KUKA KRL program: MyProgram_343().src

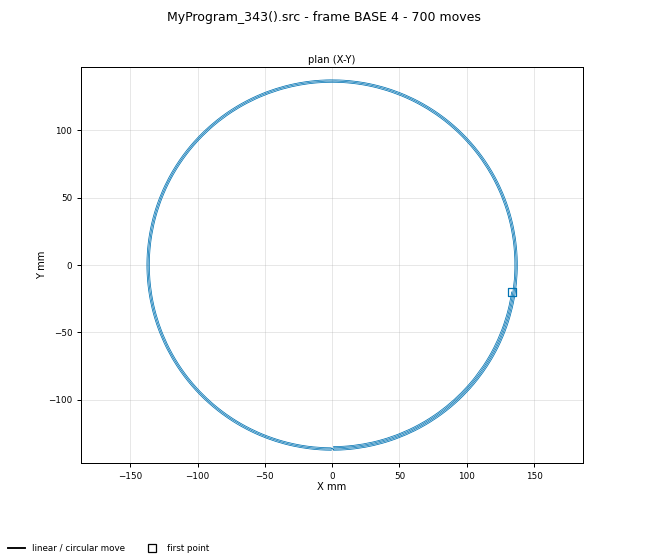
[picture p0: tool path of MyProgram_343().src in frame BASE 4, 700 of 700 moves have a stored position in this frame; points joined in program order, loops and branches not executed]
&ACCESS RVP
&REL 1
&PARAM TEMPLATE = C:\KRC\Roboter\Template\vorgabe
&PARAM EDITMASK = *
DEF MyProgram_343()
; ---- Setting reference (Base) ----
$BASE = BASE_DATA[4]

; --------------------------
; ---- Setting tool (TCP) ----
$TOOL = TOOL_DATA[3]
; --------------------------

$VEL.CP = VEL_APROX_PRINT
Startdeposition()
$VEL.CP = VEL_PRINT
LIN {X 133.4097,Y -19.9867,Z 192,A -2.4649,B 0.341,C 0.0391,E1 0.5017,E2 456.1576} C_DIS
LIN {X 132.7965,Y -23.712,Z 192,A -3.523,B 0.3407,C 0.0414,E1 0.5012,E2 457.1446} C_DIS
LIN {X 132.1464,Y -27.102,Z 192,A -4.5796,B 0.3404,C 0.0438,E1 0.5007,E2 458.1478} C_DIS
LIN {X 131.4928,Y -30.113,Z 192,A -5.5384,B 0.3401,C 0.0461,E1 0.5001,E2 459.0606} C_DIS
LIN {X 130.7303,Y -33.2675,Z 192,A -6.5628,B 0.3398,C 0.0485,E1 0.4994,E2 460.0383} C_DIS
LIN {X 129.6611,Y -37.224,Z 192,A -8.2205,B 0.3391,C 0.0529,E1 0.4982,E2 461.6861} C_DIS
LIN {X 128.1882,Y -42.0156,Z 192,A -9.2749,B 0.3388,C 0.0545,E1 0.4974,E2 462.5958} C_DIS
LIN {X 128.1882,Y -42.0156,Z 192,A -9.2759,B 0.3388,C 0.0545,E1 0.4974,E2 462.597} C_DIS
LIN {X 127.3782,Y -44.4067,Z 192,A -10.1216,B 0.3385,C 0.0565,E1 0.4967,E2 463.4123} C_DIS
LIN {X 126.1586,Y -47.7633,Z 192,A -11.2932,B 0.338,C 0.0593,E1 0.4956,E2 464.5374} C_DIS
LIN {X 124.0709,Y -52.952,Z 192,A -12.8743,B 0.3374,C 0.0626,E1 0.494,E2 466.01} C_DIS
LIN {X 123.0104,Y -55.3681,Z 192,A -13.7566,B 0.3371,C 0.0646,E1 0.493,E2 466.8596} C_DIS
LIN {X 121.4923,Y -58.6258,Z 192,A -14.8426,B 0.3366,C 0.067,E1 0.4918,E2 467.885} C_DIS
LIN {X 120.0893,Y -61.4469,Z 192,A -15.8424,B 0.3361,C 0.0692,E1 0.4906,E2 468.8379} C_DIS
LIN {X 118.1177,Y -65.1605,Z 192,A -17.0866,B 0.3356,C 0.0718,E1 0.489,E2 470.0066} C_DIS
LIN {X 116.3656,Y -68.2399,Z 192,A -18.2537,B 0.335,C 0.0745,E1 0.4874,E2 471.1268} C_DIS
LIN {X 114.2512,Y -71.7244,Z 192,A -19.5385,B 0.3344,C 0.0772,E1 0.4856,E2 472.3489} C_DIS
LIN {X 112.1427,Y -74.9777,Z 192,A -20.853,B 0.3337,C 0.0802,E1 0.4836,E2 473.6169} C_DIS
LIN {X 106.0971,Y -83.3128,Z 192,A -23.783,B 0.3323,C 0.0858,E1 0.479,E2 476.3404} C_DIS
LIN {X 106.0971,Y -83.3128,Z 192,A -23.7843,B 0.3323,C 0.0858,E1 0.479,E2 476.3418} C_DIS
LIN {X 104.2045,Y -85.6691,Z 192,A -25.3414,B 0.3312,C 0.09,E1 0.4761,E2 477.9401} C_DIS
LIN {X 100.7876,Y -89.6642,Z 192,A -26.4298,B 0.3308,C 0.0913,E1 0.4744,E2 478.862} C_DIS
LIN {X 95.9398,Y -94.8329,Z 192,A -28.8625,B 0.3294,C 0.0964,E1 0.4697,E2 481.2118} C_DIS
LIN {X 90.6247,Y -99.9239,Z 192,A -31.0205,B 0.3282,C 0.1003,E1 0.4655,E2 483.2275} C_DIS
LIN {X 90.6247,Y -99.9239,Z 192,A -31.0215,B 0.3282,C 0.1003,E1 0.4655,E2 483.2287} C_DIS
LIN {X 84.7075,Y -104.9869,Z 192,A -33.3755,B 0.3269,C 0.1046,E1 0.4607,E2 485.4418} C_DIS
LIN {X 81.036,Y -107.8465,Z 192,A -35.0547,B 0.3258,C 0.1079,E1 0.4569,E2 487.0775} C_DIS
LIN {X 78.9876,Y -109.3556,Z 192,A -35.9773,B 0.3252,C 0.1098,E1 0.4548,E2 487.9771} C_DIS
LIN {X 75.7275,Y -111.6377,Z 192,A -37.1784,B 0.3245,C 0.1118,E1 0.4521,E2 489.1052} C_DIS
LIN {X 72.4354,Y -113.8019,Z 192,A -38.5563,B 0.3236,C 0.1144,E1 0.4488,E2 490.4393} C_DIS
LIN {X 68.9662,Y -115.9366,Z 192,A -39.9703,B 0.3227,C 0.117,E1 0.4453,E2 491.8063} C_DIS
LIN {X 64.2775,Y -118.6008,Z 192,A -41.6506,B 0.3217,C 0.1197,E1 0.4413,E2 493.3947} C_DIS
LIN {X 60.7229,Y -120.4578,Z 192,A -42.8581,B 0.321,C 0.1215,E1 0.4383,E2 494.5271} C_DIS
LIN {X 57.4307,Y -122.0632,Z 192,A -44.0659,B 0.3202,C 0.1235,E1 0.4352,E2 495.6824} C_DIS
LIN {X 50.0734,Y -125.2593,Z 192,A -46.7069,B 0.3186,C 0.1276,E1 0.4283,E2 498.2071} C_DIS
LIN {X 50.0734,Y -125.2593,Z 192,A -46.7078,B 0.3186,C 0.1276,E1 0.4283,E2 498.2082} C_DIS
LIN {X 47.1757,Y -126.3787,Z 192,A -48.0353,B 0.3176,C 0.13,E1 0.4246,E2 499.5382} C_DIS
LIN {X 43.7279,Y -127.6136,Z 192,A -48.994,B 0.3172,C 0.131,E1 0.4222,E2 500.4049} C_DIS
LIN {X 40.7461,Y -128.5962,Z 192,A -50.0322,B 0.3166,C 0.1325,E1 0.4193,E2 501.398} C_DIS
LIN {X 37.4145,Y -129.6053,Z 192,A -51.21,B 0.3159,C 0.1342,E1 0.4161,E2 502.5299} C_DIS
LIN {X 34.0407,Y -130.5332,Z 192,A -52.5816,B 0.315,C 0.1363,E1 0.4121,E2 503.8847} C_DIS
LIN {X 29.855,Y -131.5518,Z 192,A -53.9027,B 0.3143,C 0.1379,E1 0.4085,E2 505.1273} C_DIS
LIN {X 26.0627,Y -132.3573,Z 192,A -55.1894,B 0.3136,C 0.1395,E1 0.4048,E2 506.3585} C_DIS
LIN {X 23.0754,Y -132.9104,Z 192,A -56.4574,B 0.3127,C 0.1414,E1 0.401,E2 507.6241} C_DIS
LIN {X 15.7245,Y -133.9776,Z 192,A -58.8527,B 0.3115,C 0.1441,E1 0.3942,E2 509.9018} C_DIS
LIN {X 11.9014,Y -134.3721,Z 192,A -60.2545,B 0.3107,C 0.1457,E1 0.39,E2 511.2683} C_DIS
LIN {X 8.165,Y -134.6498,Z 192,A -61.9084,B 0.3097,C 0.1479,E1 0.3849,E2 512.9333} C_DIS
LIN {X 3.8703,Y -134.8416,Z 192,A -63.1019,B 0.3093,C 0.1488,E1 0.3816,E2 514.0278} C_DIS
LIN {X 0.9691,Y -134.8866,Z 192,A -64.1734,B 0.3087,C 0.1499,E1 0.3784,E2 515.0745} C_DIS
Enddeposition()
LIN {X 0.9691,Y -134.8866,Z 192,A -64.1736,B 0.3087,C 0.1499,E1 0.3784,E2 515.0747} C_DIS
Startdeposition()
$VEL.CP = VEL_PRINT
LIN {X 1.4725,Y -135.79,Z 192,A -62.6899,B 0.3103,C 0.1468,E1 0.3836,E2 513.3947} C_DIS
LIN {X 7.8993,Y -135.5668,Z 192,A -61.1752,B 0.3106,C 0.1461,E1 0.3876,E2 512.0712} C_DIS
LIN {X 16.0493,Y -134.8442,Z 192,A -58.2123,B 0.3122,C 0.1426,E1 0.3964,E2 509.1841} C_DIS
LIN {X 22.9024,Y -133.8518,Z 192,A -55.8253,B 0.3135,C 0.1397,E1 0.4033,E2 506.8804} C_DIS
LIN {X 26.655,Y -133.1548,Z 192,A -54.5377,B 0.3143,C 0.1381,E1 0.407,E2 505.6431} C_DIS
LIN {X 31.7286,Y -132.037,Z 192,A -52.8298,B 0.3152,C 0.1359,E1 0.4118,E2 504.0106} C_DIS
LIN {X 34.8365,Y -131.2513,Z 192,A -51.7383,B 0.3159,C 0.1344,E1 0.4149,E2 502.9596} C_DIS
LIN {X 38.0279,Y -130.3624,Z 192,A -50.6047,B 0.3165,C 0.1328,E1 0.418,E2 501.8667} C_DIS
LIN {X 41.3599,Y -129.3438,Z 192,A -49.453,B 0.3172,C 0.1311,E1 0.4212,E2 500.7643} C_DIS
LIN {X 44.8211,Y -128.1859,Z 192,A -48.1394,B 0.3181,C 0.129,E1 0.4248,E2 499.4852} C_DIS
LIN {X 48.3933,Y -126.8826,Z 192,A -46.977,B 0.3187,C 0.1274,E1 0.4279,E2 498.3913} C_DIS
LIN {X 56.4469,Y -123.5092,Z 192,A -44.13,B 0.3204,C 0.123,E1 0.4353,E2 495.6732} C_DIS
LIN {X 56.4469,Y -123.5092,Z 192,A -44.131,B 0.3204,C 0.123,E1 0.4353,E2 495.6743} C_DIS
LIN {X 59.7456,Y -121.9467,Z 192,A -42.8805,B 0.3212,C 0.1209,E1 0.4385,E2 494.468} C_DIS
LIN {X 62.833,Y -120.3849,Z 192,A -41.7602,B 0.3219,C 0.1191,E1 0.4413,E2 493.3995} C_DIS
LIN {X 66.0403,Y -118.6581,Z 192,A -40.0165,B 0.3233,C 0.1153,E1 0.4459,E2 491.6221} C_DIS
LIN {X 71.1924,Y -115.6402,Z 192,A -38.6304,B 0.3239,C 0.1137,E1 0.4489,E2 490.4108} C_DIS
LIN {X 74.6132,Y -113.463,Z 192,A -37.2959,B 0.3247,C 0.1113,E1 0.452,E2 489.1331} C_DIS
LIN {X 77.4077,Y -111.5753,Z 192,A -36.1601,B 0.3254,C 0.1092,E1 0.4547,E2 488.0404} C_DIS
LIN {X 82.5823,Y -107.8014,Z 192,A -34.1686,B 0.3266,C 0.1057,E1 0.4591,E2 486.1562} C_DIS
LIN {X 85.9916,Y -105.1019,Z 192,A -32.4048,B 0.3278,C 0.1018,E1 0.463,E2 484.4018} C_DIS
LIN {X 89.8149,Y -101.8542,Z 192,A -31.1123,B 0.3284,C 0.0998,E1 0.4656,E2 483.2336} C_DIS
LIN {X 93.4233,Y -98.5553,Z 192,A -29.6342,B 0.3292,C 0.0971,E1 0.4685,E2 481.8427} C_DIS
LIN {X 96.6026,Y -95.4412,Z 192,A -28.4121,B 0.3299,C 0.095,E1 0.4708,E2 480.7182} C_DIS
LIN {X 100.2938,Y -91.5539,Z 192,A -26.5319,B 0.331,C 0.0909,E1 0.4744,E2 478.8935} C_DIS
LIN {X 104.4143,Y -86.8256,Z 192,A -24.5688,B 0.3321,C 0.087,E1 0.4779,E2 477.0305} C_DIS
LIN {X 106.2823,Y -84.5283,Z 192,A -23.3438,B 0.3328,C 0.084,E1 0.48,E2 475.8081} C_DIS
LIN {X 109.1526,Y -80.7877,Z 192,A -22.17,B 0.3333,C 0.082,E1 0.4818,E2 474.7539} C_DIS
LIN {X 113.2137,Y -74.9917,Z 192,A -19.9732,B 0.3344,C 0.0774,E1 0.4852,E2 472.6709} C_DIS
LIN {X 115.5535,Y -71.3337,Z 192,A -18.7754,B 0.3349,C 0.0751,E1 0.4868,E2 471.5643} C_DIS
LIN {X 117.7172,Y -67.7035,Z 192,A -17.3438,B 0.3357,C 0.0718,E1 0.4888,E2 470.1824} C_DIS
LIN {X 119.6857,Y -64.1585,Z 192,A -16.0569,B 0.3363,C 0.069,E1 0.4905,E2 468.9554} C_DIS
LIN {X 121.5238,Y -60.6031,Z 192,A -15.0058,B 0.3367,C 0.067,E1 0.4917,E2 467.9947} C_DIS
LIN {X 123.1566,Y -57.2094,Z 192,A -13.8117,B 0.3372,C 0.0643,E1 0.4931,E2 466.8557} C_DIS
LIN {X 124.7133,Y -53.7311,Z 192,A -12.1377,B 0.338,C 0.0597,E1 0.495,E2 465.1711} C_DIS
LIN {X 126.7888,Y -48.6353,Z 192,A -10.9268,B 0.3383,C 0.0578,E1 0.496,E2 464.1157} C_DIS
LIN {X 129.6598,Y -40.3634,Z 192,A -8.234,B 0.3393,C 0.0518,E1 0.4984,E2 461.5603} C_DIS
LIN {X 129.6598,Y -40.3634,Z 192,A -8.2351,B 0.3393,C 0.0518,E1 0.4984,E2 461.5615} C_DIS
LIN {X 130.6302,Y -37.1015,Z 192,A -7.1662,B 0.3397,C 0.0493,E1 0.4991,E2 460.5423} C_DIS
LIN {X 131.5427,Y -33.7207,Z 192,A -6.1536,B 0.34,C 0.047,E1 0.4998,E2 459.5926} C_DIS
LIN {X 132.3605,Y -30.351,Z 192,A -5.0792,B 0.3404,C 0.0445,E1 0.5005,E2 458.5702} C_DIS
LIN {X 133.111,Y -26.8701,Z 192,A -3.9875,B 0.3407,C 0.042,E1 0.5011,E2 457.5333} C_DIS
LIN {X 133.867,Y -22.8113,Z 192,A -2.6959,B 0.341,C 0.039,E1 0.5017,E2 456.3014} C_DIS
LIN {X 134.4202,Y -19.2804,Z 192,A -1.692,B 0.3413,C 0.0368,E1 0.5021,E2 455.3639} C_DIS
LIN {X 135.3511,Y -10.9921,Z 192,A 0.9276,B 0.3419,C 0.0306,E1 0.5028,E2 452.8614} C_DIS
LIN {X 135.5771,Y -7.7314,Z 192,A 2.3132,B 0.3422,C 0.0267,E1 0.503,E2 451.4743} C_DIS
LIN {X 135.7734,Y -2.4939,Z 192,A 3.3682,B 0.3423,C 0.0251,E1 0.503,E2 450.5685} C_DIS
LIN {X 135.7363,Y 4.038,Z 192,A 5.4733,B 0.3427,C 0.0199,E1 0.503,E2 448.5455} C_DIS
LIN {X 135.5506,Y 8.1615,Z 192,A 6.7874,B 0.3428,C 0.0167,E1 0.5028,E2 447.2848} C_DIS
LIN {X 135.0975,Y 13.7679,Z 192,A 8.6876,B 0.343,C 0.0119,E1 0.5023,E2 445.443} C_DIS
LIN {X 134.622,Y 17.8179,Z 192,A 9.6568,B 0.3431,C 0.0101,E1 0.502,E2 444.5665} C_DIS
LIN {X 133.9777,Y 22.1475,Z 192,A 10.9665,B 0.3431,C 0.007,E1 0.5015,E2 443.322} C_DIS
LIN {X 133.1461,Y 26.6974,Z 192,A 12.3466,B 0.3432,C 0.0037,E1 0.5008,E2 442.0106} C_DIS
LIN {X 132.4245,Y 30.0708,Z 192,A 13.3988,B 0.3432,C 0.0013,E1 0.5002,E2 441.0063} C_DIS
LIN {X 131.5924,Y 33.5252,Z 192,A 14.4549,B 0.3432,C -0.0012,E1 0.4995,E2 440.0026} C_DIS
LIN {X 130.641,Y 37.0629,Z 192,A 15.6611,B 0.3432,C -0.0042,E1 0.4986,E2 438.8361} C_DIS
LIN {X 129.434,Y 41.0773,Z 192,A 16.8602,B 0.3432,C -0.0069,E1 0.4977,E2 437.7032} C_DIS
LIN {X 128.3363,Y 44.3873,Z 192,A 17.8557,B 0.3432,C -0.0091,E1 0.4968,E2 436.7624} C_DIS
LIN {X 125.7972,Y 51.1436,Z 192,A 20.1438,B 0.3429,C -0.0146,E1 0.4946,E2 434.5603} C_DIS
LIN {X 124.4817,Y 54.2669,Z 192,A 21.546,B 0.3428,C -0.0184,E1 0.493,E2 433.1609} C_DIS
LIN {X 122.3912,Y 58.8295,Z 192,A 22.6661,B 0.3426,C -0.0204,E1 0.4918,E2 432.1522} C_DIS
LIN {X 120.4119,Y 62.7817,Z 192,A 23.9979,B 0.3425,C -0.0235,E1 0.4902,E2 430.8788} C_DIS
LIN {X 118.3975,Y 66.5056,Z 192,A 25.2069,B 0.3423,C -0.0262,E1 0.4886,E2 429.7323} C_DIS
LIN {X 115.3361,Y 71.6837,Z 192,A 27.0194,B 0.3419,C -0.0302,E1 0.4861,E2 427.9972} C_DIS
LIN {X 115.3361,Y 71.6837,Z 192,A 27.0182,B 0.3419,C -0.0302,E1 0.4861,E2 427.9986} C_DIS
LIN {X 111.0879,Y 78.1055,Z 192,A 29.5384,B 0.3413,C -0.0361,E1 0.4823,E2 425.5547} C_DIS
LIN {X 111.0879,Y 78.1055,Z 192,A 29.5372,B 0.3413,C -0.0361,E1 0.4823,E2 425.556} C_DIS
LIN {X 108.4803,Y 81.6884,Z 192,A 30.8927,B 0.341,C -0.0392,E1 0.48,E2 424.2536} C_DIS
LIN {X 105.7497,Y 85.1937,Z 192,A 32.2508,B 0.3407,C -0.0422,E1 0.4777,E2 422.948} C_DIS
LIN {X 102.9151,Y 88.5971,Z 192,A 33.6229,B 0.3403,C -0.0452,E1 0.4753,E2 421.6259} C_DIS
LIN {X 99.8987,Y 91.9849,Z 192,A 35.0225,B 0.3398,C -0.0483,E1 0.4727,E2 420.2773} C_DIS
LIN {X 96.841,Y 95.1987,Z 192,A 36.3962,B 0.3394,C -0.0512,E1 0.47,E2 418.9523} C_DIS
LIN {X 93.6737,Y 98.317,Z 192,A 37.7131,B 0.339,C -0.054,E1 0.4674,E2 417.6895} C_DIS
LIN {X 90.8265,Y 100.9534,Z 192,A 39.0052,B 0.3385,C -0.0568,E1 0.4647,E2 416.4302} C_DIS
LIN {X 87.3782,Y 103.952,Z 192,A 40.4055,B 0.338,C -0.0597,E1 0.4618,E2 415.0798} C_DIS
LIN {X 83.9483,Y 106.741,Z 192,A 41.7906,B 0.3375,C -0.0625,E1 0.4587,E2 413.7393} C_DIS
LIN {X 80.4014,Y 109.4375,Z 192,A 43.1692,B 0.337,C -0.0653,E1 0.4556,E2 412.4066} C_DIS
LIN {X 76.908,Y 111.9202,Z 192,A 44.5345,B 0.3364,C -0.068,E1 0.4524,E2 411.0814} C_DIS
LIN {X 70.7158,Y 115.9326,Z 192,A 47.4997,B 0.3351,C -0.0744,E1 0.4451,E2 408.1298} C_DIS
LIN {X 64.99,Y 119.2362,Z 192,A 48.9607,B 0.3346,C -0.0765,E1 0.4417,E2 406.7851} C_DIS
LIN {X 64.99,Y 119.2362,Z 192,A 48.9597,B 0.3346,C -0.0765,E1 0.4417,E2 406.7862} C_DIS
LIN {X 61.8234,Y 120.9063,Z 192,A 50.0685,B 0.3341,C -0.0786,E1 0.4388,E2 405.7115} C_DIS
LIN {X 58.7094,Y 122.4486,Z 192,A 51.1303,B 0.3337,C -0.0805,E1 0.4361,E2 404.6839} C_DIS
LIN {X 55.145,Y 124.0949,Z 192,A 52.7437,B 0.3329,C -0.0837,E1 0.4318,E2 403.0743} C_DIS
LIN {X 51.4888,Y 125.658,Z 192,A 53.7858,B 0.3325,C -0.0853,E1 0.429,E2 402.0849} C_DIS
LIN {X 44.4612,Y 128.3107,Z 192,A 56.2033,B 0.3314,C -0.0894,E1 0.4225,E2 399.7283} C_DIS
LIN {X 40.3327,Y 129.6692,Z 192,A 57.6658,B 0.3307,C -0.0918,E1 0.4183,E2 398.2954} C_DIS
LIN {X 36.6706,Y 130.7507,Z 192,A 58.8285,B 0.3302,C -0.0936,E1 0.4151,E2 397.1677} C_DIS
LIN {X 33.7939,Y 131.5242,Z 192,A 59.8669,B 0.3298,C -0.0953,E1 0.4121,E2 396.1463} C_DIS
LIN {X 30.415,Y 132.3459,Z 192,A 61.0053,B 0.3293,C -0.097,E1 0.4088,E2 395.0332} C_DIS
LIN {X 27.1208,Y 133.06,Z 192,A 62.1582,B 0.3287,C -0.0988,E1 0.4055,E2 393.9007} C_DIS
LIN {X 23.1296,Y 133.8139,Z 192,A 63.4762,B 0.3282,C -0.1006,E1 0.4016,E2 392.6126} C_DIS
LIN {X 18.7384,Y 134.4976,Z 192,A 65.0518,B 0.3275,C -0.1029,E1 0.397,E2 391.0593} C_DIS
LIN {X 14.8354,Y 134.9835,Z 192,A 66.3029,B 0.327,C -0.1045,E1 0.3933,E2 389.838} C_DIS
LIN {X 11.464,Y 135.3112,Z 192,A 67.7711,B 0.3263,C -0.1066,E1 0.3888,E2 388.3675} C_DIS
LIN {X 8.0751,Y 135.556,Z 192,A 69.1287,B 0.3257,C -0.1084,E1 0.3847,E2 387.0158} C_DIS
LIN {X 3.576,Y 135.7491,Z 192,A 70.2654,B 0.3253,C -0.1095,E1 0.3813,E2 385.9331} C_DIS
LIN {X 0.1229,Y 135.7975,Z 192,A 71.9806,B 0.3246,C -0.1118,E1 0.376,E2 384.2007} C_DIS
LIN {X -4.7497,Y 135.714,Z 192,A 73.1804,B 0.3242,C -0.1128,E1 0.3725,E2 383.0603} C_DIS
LIN {X -11.1773,Y 135.3354,Z 192,A 75.4863,B 0.3234,C -0.1151,E1 0.3655,E2 380.7826} C_DIS
LIN {X -11.1773,Y 135.3354,Z 192,A 75.4853,B 0.3234,C -0.1151,E1 0.3655,E2 380.7837} C_DIS
LIN {X -14.4957,Y 135.02,Z 192,A 76.7242,B 0.323,C -0.1163,E1 0.3616,E2 379.5564} C_DIS
LIN {X -18.0871,Y 134.5867,Z 192,A 78.2157,B 0.3225,C -0.1176,E1 0.357,E2 378.0679} C_DIS
LIN {X -23.7428,Y 133.7042,Z 192,A 80.1421,B 0.3219,C -0.1191,E1 0.3512,E2 376.1739} C_DIS
LIN {X -26.8096,Y 133.1233,Z 192,A 81.2932,B 0.3216,C -0.1199,E1 0.3477,E2 375.034} C_DIS
LIN {X -30.1125,Y 132.415,Z 192,A 82.5489,B 0.3213,C -0.1208,E1 0.3439,E2 373.7895} C_DIS
LIN {X -33.0981,Y 131.7008,Z 192,A 83.7349,B 0.321,C -0.1215,E1 0.3403,E2 372.611} C_DIS
LIN {X -36.3353,Y 130.8445,Z 192,A 85.0496,B 0.3207,C -0.1223,E1 0.3364,E2 371.303} C_DIS
LIN {X -39.8506,Y 129.8168,Z 192,A 86.3814,B 0.3205,C -0.1229,E1 0.3324,E2 369.985} C_DIS
LIN {X -47.1065,Y 127.3645,Z 192,A 89.4772,B 0.32,C -0.1242,E1 0.3232,E2 366.8992} C_DIS
LIN {X -50.5062,Y 126.0541,Z 192,A 90.8198,B 0.3199,C -0.1245,E1 0.3193,E2 365.5691} C_DIS
LIN {X -53.4792,Y 124.8223,Z 192,A 92.1446,B 0.3197,C -0.1249,E1 0.3155,E2 364.2468} C_DIS
LIN {X -56.5005,Y 123.4844,Z 192,A 93.6692,B 0.3197,C -0.1252,E1 0.3111,E2 362.715} C_DIS
LIN {X -60.1379,Y 121.7532,Z 192,A 95.1103,B 0.3196,C -0.1252,E1 0.307,E2 361.2902} C_DIS
LIN {X -62.8614,Y 120.37,Z 192,A 96.4981,B 0.3196,C -0.1253,E1 0.3031,E2 359.897} C_DIS
LIN {X -65.1407,Y 119.154,Z 192,A 98.2018,B 0.3196,C -0.1254,E1 0.2983,E2 358.1562} C_DIS
LIN {X -69.1565,Y 116.8697,Z 192,A 100.5286,B 0.3196,C -0.1252,E1 0.2919,E2 355.8066} C_DIS
LIN {X -74.392,Y 113.6086,Z 192,A 102.4653,B 0.3199,C -0.1244,E1 0.2869,E2 353.9127} C_DIS
LIN {X -78.1055,Y 111.0879,Z 192,A 104.3444,B 0.3202,C -0.1238,E1 0.282,E2 352.0353} C_DIS
LIN {X -84.2675,Y 106.4898,Z 192,A 108.0185,B 0.3208,C -0.1221,E1 0.2728,E2 348.3361} C_DIS
LIN {X -87.7024,Y 103.6791,Z 192,A 110.1144,B 0.3213,C -0.1208,E1 0.2677,E2 346.227} C_DIS
LIN {X -90.5619,Y 101.1904,Z 192,A 112.1309,B 0.3218,C -0.1194,E1 0.2629,E2 344.1846} C_DIS
LIN {X -96.1175,Y 95.9295,Z 192,A 115.7507,B 0.323,C -0.1163,E1 0.2547,E2 340.5407} C_DIS
LIN {X -99.6018,Y 92.3068,Z 192,A 118.9115,B 0.324,C -0.1133,E1 0.2479,E2 337.3112} C_DIS
LIN {X -102.7604,Y 88.7767,Z 192,A 121.1506,B 0.3249,C -0.1107,E1 0.2433,E2 335.0564} C_DIS
LIN {X -105.1673,Y 85.9115,Z 192,A 122.7645,B 0.3256,C -0.1087,E1 0.2402,E2 333.4407} C_DIS
LIN {X -107.9808,Y 82.3477,Z 192,A 125.1208,B 0.3266,C -0.1056,E1 0.2357,E2 331.0545} C_DIS
LIN {X -110.4857,Y 78.9549,Z 192,A 127.5551,B 0.3277,C -0.1022,E1 0.2312,E2 328.5741} C_DIS
LIN {X -112.8828,Y 75.4881,Z 192,A 130.0053,B 0.3288,C -0.0986,E1 0.227,E2 326.0753} C_DIS
LIN {X -115.39,Y 71.5971,Z 192,A 132.5678,B 0.33,C -0.0945,E1 0.2228,E2 323.4679} C_DIS
LIN {X -117.9533,Y 67.2903,Z 192,A 135.6435,B 0.3314,C -0.0893,E1 0.218,E2 320.3187} C_DIS
LIN {X -117.9533,Y 67.2903,Z 192,A 135.6426,B 0.3314,C -0.0893,E1 0.218,E2 320.3197} C_DIS
LIN {X -119.8647,Y 63.8237,Z 192,A 138.2995,B 0.3327,C -0.0846,E1 0.2141,E2 317.5845} C_DIS
LIN {X -119.8647,Y 63.8237,Z 192,A 138.2983,B 0.3327,C -0.0846,E1 0.2141,E2 317.5858} C_DIS
LIN {X -121.8013,Y 60.0404,Z 192,A 140.6505,B 0.3338,C -0.0801,E1 0.2109,E2 315.1883} C_DIS
LIN {X -123.2085,Y 57.0972,Z 192,A 142.6988,B 0.3347,C -0.0761,E1 0.2083,E2 313.0841} C_DIS
LIN {X -124.9738,Y 53.1288,Z 192,A 145.7,B 0.336,C -0.07,E1 0.2047,E2 309.9827} C_DIS
LIN {X -124.9738,Y 53.1288,Z 192,A 145.6985,B 0.336,C -0.07,E1 0.2047,E2 309.9843} C_DIS
LIN {X -126.4123,Y 49.6038,Z 192,A 148.0693,B 0.3371,C -0.0649,E1 0.202,E2 307.546} C_DIS
LIN {X -127.7059,Y 46.1697,Z 192,A 150.5189,B 0.338,C -0.0596,E1 0.1995,E2 305.0146} C_DIS
LIN {X -127.7059,Y 46.1697,Z 192,A 150.5179,B 0.338,C -0.0596,E1 0.1995,E2 305.0157} C_DIS
LIN {X -128.8341,Y 42.9211,Z 192,A 152.7094,B 0.3389,C -0.0547,E1 0.1974,E2 302.7555} C_DIS
LIN {X -129.8022,Y 39.8984,Z 192,A 154.9878,B 0.3397,C -0.0494,E1 0.1953,E2 300.3876} C_DIS
LIN {X -129.8022,Y 39.8984,Z 192,A 154.9867,B 0.3397,C -0.0494,E1 0.1953,E2 300.3888} C_DIS
LIN {X -130.7106,Y 36.8139,Z 192,A 157.2197,B 0.3404,C -0.0442,E1 0.1935,E2 298.0703} C_DIS
LIN {X -130.7106,Y 36.8139,Z 192,A 157.2187,B 0.3404,C -0.0442,E1 0.1935,E2 298.0714} C_DIS
LIN {X -131.6889,Y 33.1448,Z 192,A 160.4515,B 0.3413,C -0.0365,E1 0.1911,E2 294.6736} C_DIS
LIN {X -132.445,Y 29.9813,Z 192,A 162.4614,B 0.3418,C -0.0316,E1 0.1898,E2 292.5976} C_DIS
LIN {X -132.445,Y 29.9813,Z 192,A 162.4597,B 0.3418,C -0.0316,E1 0.1898,E2 292.5995} C_DIS
LIN {X -133.33,Y 25.7622,Z 192,A 165.3538,B 0.3424,C -0.0243,E1 0.1881,E2 289.5915} C_DIS
LIN {X -133.33,Y 25.7622,Z 192,A 165.3524,B 0.3424,C -0.0243,E1 0.1881,E2 289.5931} C_DIS
LIN {X -133.8722,Y 22.7799,Z 192,A 167.7024,B 0.3428,C -0.0184,E1 0.1869,E2 287.1263} C_DIS
LIN {X -133.8722,Y 22.7799,Z 192,A 167.7005,B 0.3428,C -0.0184,E1 0.1869,E2 287.1284} C_DIS
LIN {X -134.4634,Y 18.9781,Z 192,A 170.4332,B 0.3431,C -0.0114,E1 0.1857,E2 284.2721} C_DIS
LIN {X -134.4634,Y 18.9781,Z 192,A 170.4315,B 0.3431,C -0.0114,E1 0.1857,E2 284.2739} C_DIS
LIN {X -134.9487,Y 15.1585,Z 192,A 173.4823,B 0.3432,C -0.0036,E1 0.1847,E2 281.0595} C_DIS
LIN {X -134.9487,Y 15.1585,Z 192,A 173.4795,B 0.3432,C -0.0036,E1 0.1847,E2 281.0626} C_DIS
LIN {X -135.3338,Y 11.1966,Z 192,A 176.3421,B 0.3432,C 0.0038,E1 0.1839,E2 278.0606} C_DIS
LIN {X -135.3338,Y 11.1966,Z 192,A 176.34,B 0.3432,C 0.0038,E1 0.1839,E2 278.063} C_DIS
LIN {X -135.6201,Y 6.9103,Z 192,A 179.4355,B 0.343,C 0.0119,E1 0.1834,E2 274.8127} C_DIS
LIN {X -135.6201,Y 6.9103,Z 192,A 179.4334,B 0.343,C 0.0119,E1 0.1834,E2 274.815} C_DIS
LIN {X -135.7595,Y 3.2026,Z 192,A -177.5746,B 0.3427,C 0.0197,E1 0.1831,E2 271.6464} C_DIS
LIN {X -135.7595,Y 3.2026,Z 192,A -177.5775,B 0.3427,C 0.0197,E1 0.1831,E2 271.6497} C_DIS
LIN {X -135.7975,Y -0.3872,Z 192,A -174.886,B 0.3422,C 0.0267,E1 0.1831,E2 268.8092} C_DIS
LIN {X -135.7975,Y -0.3872,Z 192,A -174.8886,B 0.3422,C 0.0267,E1 0.1831,E2 268.8122} C_DIS
LIN {X -135.7197,Y -4.6055,Z 192,A -171.8245,B 0.3415,C 0.0347,E1 0.1834,E2 265.5821} C_DIS
LIN {X -135.7197,Y -4.6055,Z 192,A -171.8269,B 0.3415,C 0.0347,E1 0.1834,E2 265.5847} C_DIS
LIN {X -135.5466,Y -8.2274,Z 192,A -169.3151,B 0.3408,C 0.0412,E1 0.1837,E2 262.9438} C_DIS
LIN {X -135.5466,Y -8.2274,Z 192,A -169.3164,B 0.3408,C 0.0412,E1 0.1837,E2 262.9452} C_DIS
LIN {X -135.3293,Y -11.2493,Z 192,A -166.9224,B 0.34,C 0.0473,E1 0.1843,E2 260.4019} C_DIS
LIN {X -135.3293,Y -11.2493,Z 192,A -166.9241,B 0.34,C 0.0473,E1 0.1843,E2 260.4038} C_DIS
LIN {X -134.9468,Y -15.1761,Z 192,A -163.8815,B 0.3388,C 0.055,E1 0.1853,E2 257.1734} C_DIS
LIN {X -134.9468,Y -15.1761,Z 192,A -163.884,B 0.3388,C 0.055,E1 0.1853,E2 257.1763} C_DIS
LIN {X -134.4347,Y -19.1791,Z 192,A -161.193,B 0.3377,C 0.0618,E1 0.1863,E2 254.3486} C_DIS
LIN {X -134.4347,Y -19.1791,Z 192,A -161.1942,B 0.3377,C 0.0618,E1 0.1863,E2 254.35} C_DIS
LIN {X -133.9536,Y -22.2921,Z 192,A -158.8015,B 0.3365,C 0.0676,E1 0.1875,E2 251.8079} C_DIS
LIN {X -133.9536,Y -22.2921,Z 192,A -158.8029,B 0.3365,C 0.0676,E1 0.1875,E2 251.8095} C_DIS
LIN {X -133.2691,Y -26.0805,Z 192,A -155.9622,B 0.3351,C 0.0744,E1 0.189,E2 248.7957} C_DIS
LIN {X -133.2691,Y -26.0805,Z 192,A -155.964,B 0.3351,C 0.0744,E1 0.189,E2 248.7978} C_DIS
LIN {X -132.4319,Y -30.0387,Z 192,A -153.3172,B 0.3336,C 0.0807,E1 0.1907,E2 246.0156} C_DIS
LIN {X -132.4319,Y -30.0387,Z 192,A -153.3182,B 0.3336,C 0.0807,E1 0.1907,E2 246.0168} C_DIS
LIN {X -131.6604,Y -33.2572,Z 192,A -150.9302,B 0.3322,C 0.0862,E1 0.1924,E2 243.4842} C_DIS
LIN {X -131.6604,Y -33.2572,Z 192,A -150.9312,B 0.3322,C 0.0862,E1 0.1924,E2 243.4854} C_DIS
LIN {X -130.6807,Y -36.9208,Z 192,A -148.264,B 0.3306,C 0.0922,E1 0.1946,E2 240.6609} C_DIS
LIN {X -130.6807,Y -36.9208,Z 192,A -148.2651,B 0.3306,C 0.0922,E1 0.1946,E2 240.6623} C_DIS
LIN {X -129.4697,Y -40.9657,Z 192,A -145.6057,B 0.3289,C 0.0981,E1 0.1969,E2 237.8724} C_DIS
LIN {X -128.5394,Y -43.8017,Z 192,A -143.0028,B 0.3273,C 0.1034,E1 0.1995,E2 235.0672} C_DIS
LIN {X -128.5394,Y -43.8017,Z 192,A -143.005,B 0.3273,C 0.1034,E1 0.1995,E2 235.0697} C_DIS
LIN {X -126.5814,Y -49.1688,Z 192,A -139.6955,B 0.3251,C 0.1102,E1 0.203,E2 231.6239} C_DIS
LIN {X -125.379,Y -52.1589,Z 192,A -137.6043,B 0.3237,C 0.1143,E1 0.2055,E2 229.4209} C_DIS
LIN {X -124.0007,Y -55.3557,Z 192,A -135.3447,B 0.3221,C 0.1185,E1 0.2083,E2 227.0397} C_DIS
LIN {X -122.6394,Y -58.3099,Z 192,A -133.3866,B 0.3208,C 0.1221,E1 0.2108,E2 224.9911} C_DIS
LIN {X -121.1396,Y -61.365,Z 192,A -131.3757,B 0.3194,C 0.1256,E1 0.2136,E2 222.8909} C_DIS
LIN {X -118.5397,Y -66.2526,Z 192,A -127.8127,B 0.3171,C 0.1314,E1 0.2189,E2 219.136} C_DIS
LIN {X -118.5397,Y -66.2526,Z 192,A -127.8139,B 0.3171,C 0.1314,E1 0.2189,E2 219.1375} C_DIS
LIN {X -116.4921,Y -69.7899,Z 192,A -125.4446,B 0.3156,C 0.135,E1 0.2227,E2 216.6668} C_DIS
LIN {X -114.1523,Y -73.5552,Z 192,A -122.8639,B 0.314,C 0.1387,E1 0.2271,E2 213.9738} C_DIS
LIN {X -111.6398,Y -77.315,Z 192,A -120.4132,B 0.3125,C 0.142,E1 0.2314,E2 211.4372} C_DIS
LIN {X -109.1955,Y -80.7309,Z 192,A -118.0198,B 0.3111,C 0.145,E1 0.2359,E2 208.9448} C_DIS
LIN {X -106.9917,Y -83.6286,Z 192,A -115.9081,B 0.31,C 0.1473,E1 0.24,E2 206.7411} C_DIS
LIN {X -103.6097,Y -87.784,Z 192,A -113.292,B 0.3087,C 0.1502,E1 0.2453,E2 204.068} C_DIS
LIN {X -100.6611,Y -91.15,Z 192,A -111.1936,B 0.3076,C 0.1523,E1 0.2496,E2 201.9358} C_DIS
LIN {X -98.0426,Y -93.9608,Z 192,A -109.0988,B 0.3067,C 0.154,E1 0.2543,E2 199.7647} C_DIS
LIN {X -93.0952,Y -98.864,Z 192,A -105.4744,B 0.3054,C 0.1566,E1 0.2626,E2 196.0295} C_DIS
LIN {X -89.0285,Y -102.5426,Z 192,A -103.0282,B 0.3046,C 0.1583,E1 0.2684,E2 193.5616} C_DIS
LIN {X -85.5635,Y -105.4514,Z 192,A -100.9801,B 0.304,C 0.1594,E1 0.2734,E2 191.4905} C_DIS
LIN {X -82.2995,Y -108.0177,Z 192,A -99.0862,B 0.3036,C 0.1602,E1 0.2781,E2 189.5732} C_DIS
LIN {X -78.9549,Y -110.4857,Z 192,A -97.2587,B 0.3032,C 0.161,E1 0.2828,E2 187.7333} C_DIS
LIN {X -74.2286,Y -113.7154,Z 192,A -94.5567,B 0.3029,C 0.1616,E1 0.29,E2 184.9841} C_DIS
LIN {X -70.9948,Y -115.7614,Z 192,A -92.7033,B 0.3028,C 0.1617,E1 0.2951,E2 183.0914} C_DIS
LIN {X -68.1048,Y -117.4849,Z 192,A -91.4805,B 0.3026,C 0.162,E1 0.2983,E2 181.9} C_DIS
LIN {X -64.1165,Y -119.7083,Z 192,A -89.4971,B 0.3026,C 0.162,E1 0.3039,E2 179.9065} C_DIS
LIN {X -60.3737,Y -121.6369,Z 192,A -87.8446,B 0.3026,C 0.162,E1 0.3085,E2 178.2734} C_DIS
LIN {X -54.7041,Y -124.2921,Z 192,A -85.1604,B 0.3028,C 0.1616,E1 0.3162,E2 175.581} C_DIS
LIN {X -51.7385,Y -125.5546,Z 192,A -83.4857,B 0.3032,C 0.1609,E1 0.3212,E2 173.8545} C_DIS
LIN {X -47.6318,Y -127.1678,Z 192,A -82.1247,B 0.3032,C 0.1609,E1 0.325,E2 172.5738} C_DIS
LIN {X -43.3537,Y -128.69,Z 192,A -80.3553,B 0.3035,C 0.1604,E1 0.3302,E2 170.8271} C_DIS
LIN {X -40.0287,Y -129.7623,Z 192,A -79.0364,B 0.3038,C 0.1599,E1 0.3341,E2 169.5325} C_DIS
LIN {X -36.7475,Y -130.7292,Z 192,A -77.6985,B 0.3041,C 0.1592,E1 0.338,E2 168.2109} C_DIS
LIN {X -33.3322,Y -131.6413,Z 192,A -76.3037,B 0.3045,C 0.1585,E1 0.3422,E2 166.8307} C_DIS
LIN {X -29.0795,Y -132.6464,Z 192,A -74.6338,B 0.305,C 0.1575,E1 0.3472,E2 165.1879} C_DIS
LIN {X -24.7209,Y -133.529,Z 192,A -72.7216,B 0.3057,C 0.156,E1 0.3531,E2 163.2686} C_DIS
LIN {X -21.3876,Y -134.1024,Z 192,A -71.666,B 0.306,C 0.1555,E1 0.3562,E2 162.2721} C_DIS
LIN {X -17.7399,Y -134.6322,Z 192,A -70.3604,B 0.3064,C 0.1546,E1 0.3601,E2 161.0059} C_DIS
LIN {X -13.7942,Y -135.0955,Z 192,A -68.8386,B 0.3071,C 0.1534,E1 0.3647,E2 159.5078} C_DIS
LIN {X -6.1085,Y -135.6604,Z 192,A -66.145,B 0.3082,C 0.1512,E1 0.3728,E2 156.9021} C_DIS
LIN {X -0.895,Y -135.7931,Z 192,A -64.1699,B 0.3092,C 0.1492,E1 0.3788,E2 154.9616} C_DIS
LIN {X -0.895,Y -135.7931,Z 192,A -64.1704,B 0.3092,C 0.1492,E1 0.3788,E2 154.9622} C_DIS
Enddeposition()
LIN {X 0.9731,Y -136.6912,Z 192,A -67.3037,B 0.3824,C 0.1585,E1 0.4442,E2 158.7118} C_DIS
Startdeposition()
$VEL.CP = VEL_PRINT
LIN {X 0.9731,Y -136.6912,Z 192,A -67.3074,B 0.3824,C 0.1585,E1 0.4442,E2 158.7162} C_DIS
LIN {X -5.7459,Y -136.5748,Z 192,A -70.0145,B 0.3814,C 0.1609,E1 0.4361,E2 161.408} C_DIS
LIN {X -10.3047,Y -136.3064,Z 192,A -71.8473,B 0.3808,C 0.1623,E1 0.4306,E2 163.229} C_DIS
LIN {X -14.1675,Y -135.9594,Z 192,A -73.1818,B 0.3805,C 0.163,E1 0.4267,E2 164.5183} C_DIS
LIN {X -19.2096,Y -135.3384,Z 192,A -75.0945,B 0.38,C 0.1641,E1 0.4211,E2 166.3977} C_DIS
LIN {X -23.0056,Y -134.7457,Z 192,A -76.8038,B 0.3795,C 0.1653,E1 0.416,E2 168.1238} C_DIS
LIN {X -28.1533,Y -133.7659,Z 192,A -78.7067,B 0.3792,C 0.166,E1 0.4105,E2 169.9811} C_DIS
LIN {X -31.674,Y -132.9749,Z 192,A -80.1004,B 0.379,C 0.1664,E1 0.4064,E2 171.3567} C_DIS
LIN {X -35.2342,Y -132.0756,Z 192,A -81.5505,B 0.3788,C 0.1669,E1 0.4022,E2 172.7934} C_DIS
LIN {X -39.0894,Y -130.9883,Z 192,A -83.1887,B 0.3786,C 0.1674,E1 0.3975,E2 174.426} C_DIS
LIN {X -42.9296,Y -129.7787,Z 192,A -84.7674,B 0.3785,C 0.1676,E1 0.393,E2 175.9881} C_DIS
LIN {X -45.8654,Y -128.7712,Z 192,A -86.0592,B 0.3784,C 0.1678,E1 0.3893,E2 177.279} C_DIS
LIN {X -48.5465,Y -127.7851,Z 192,A -88.0785,B 0.3779,C 0.1689,E1 0.3833,E2 179.4303} C_DIS
LIN {X -54.4907,Y -125.3643,Z 192,A -89.7122,B 0.3784,C 0.1678,E1 0.3792,E2 180.8964} C_DIS
LIN {X -59.2973,Y -123.164,Z 192,A -92.2684,B 0.3784,C 0.1678,E1 0.372,E2 183.5079} C_DIS
LIN {X -63.1248,Y -121.247,Z 192,A -94.0477,B 0.3785,C 0.1675,E1 0.3672,E2 185.2855} C_DIS
LIN {X -67.0584,Y -119.118,Z 192,A -96.0218,B 0.3788,C 0.167,E1 0.3619,E2 187.2761} C_DIS
LIN {X -74.0223,Y -114.9206,Z 192,A -99.3712,B 0.3794,C 0.1655,E1 0.3533,E2 190.6172} C_DIS
LIN {X -78.6907,Y -111.7752,Z 192,A -102.2169,B 0.3799,C 0.1643,E1 0.346,E2 193.5411} C_DIS
LIN {X -82.2005,Y -109.2201,Z 192,A -104.2313,B 0.3804,C 0.1631,E1 0.3411,E2 195.5869} C_DIS
LIN {X -86.184,Y -106.1056,Z 192,A -106.6437,B 0.3812,C 0.1614,E1 0.3353,E2 198.0461} C_DIS
LIN {X -89.707,Y -103.1437,Z 192,A -108.7982,B 0.3819,C 0.1597,E1 0.3303,E2 200.2366} C_DIS
LIN {X -92.1961,Y -100.9255,Z 192,A -110.9535,B 0.3825,C 0.1582,E1 0.3253,E2 202.5118} C_DIS
LIN {X -95.6748,Y -97.6332,Z 192,A -112.6984,B 0.3834,C 0.156,E1 0.3216,E2 204.2154} C_DIS
LIN {X -98.6164,Y -94.6616,Z 192,A -114.8416,B 0.3843,C 0.1539,E1 0.317,E2 206.4202} C_DIS
LIN {X -101.6502,Y -91.3959,Z 192,A -117.092,B 0.3853,C 0.1513,E1 0.3124,E2 208.7306} C_DIS
LIN {X -104.6535,Y -87.9406,Z 192,A -119.403,B 0.3864,C 0.1484,E1 0.3078,E2 211.1029} C_DIS
LIN {X -107.9374,Y -83.8776,Z 192,A -121.968,B 0.3877,C 0.145,E1 0.303,E2 213.7264} C_DIS
LIN {X -110.3917,Y -80.6209,Z 192,A -124.3215,B 0.3889,C 0.1418,E1 0.2987,E2 216.18} C_DIS
LIN {X -112.9738,Y -76.961,Z 192,A -126.7222,B 0.3902,C 0.1381,E1 0.2945,E2 218.6615} C_DIS
LIN {X -115.4029,Y -73.2681,Z 192,A -129.1374,B 0.3915,C 0.1343,E1 0.2906,E2 221.1629} C_DIS
LIN {X -117.7133,Y -69.4952,Z 192,A -131.4629,B 0.3929,C 0.1303,E1 0.287,E2 223.5604} C_DIS
LIN {X -120.1701,Y -65.1534,Z 192,A -134.5591,B 0.3946,C 0.125,E1 0.2824,E2 226.8093} C_DIS
LIN {X -122.458,Y -60.7411,Z 192,A -137.1396,B 0.3961,C 0.1201,E1 0.2789,E2 229.4644} C_DIS
LIN {X -124.0032,Y -57.5204,Z 192,A -139.1643,B 0.3973,C 0.1161,E1 0.2763,E2 231.5681} C_DIS
LIN {X -125.3003,Y -54.6387,Z 192,A -141.1058,B 0.3984,C 0.1123,E1 0.274,E2 233.6015} C_DIS
LIN {X -126.7165,Y -51.2672,Z 192,A -143.1882,B 0.3996,C 0.108,E1 0.2716,E2 235.7651} C_DIS
LIN {X -129.0099,Y -45.1887,Z 192,A -147.223,B 0.4018,C 0.0995,E1 0.2674,E2 239.9922} C_DIS
LIN {X -129.0099,Y -45.1887,Z 192,A -147.2238,B 0.4018,C 0.0995,E1 0.2674,E2 239.9932} C_DIS
LIN {X -130.0778,Y -42.0163,Z 192,A -149.111,B 0.4028,C 0.0952,E1 0.2657,E2 241.9504} C_DIS
LIN {X -131.0888,Y -38.7461,Z 192,A -151.3264,B 0.404,C 0.0903,E1 0.2638,E2 244.2782} C_DIS
LIN {X -132.4138,Y -33.9426,Z 192,A -154.4321,B 0.4055,C 0.0831,E1 0.2614,E2 247.5285} C_DIS
LIN {X -133.2699,Y -30.4065,Z 192,A -156.6861,B 0.4066,C 0.0778,E1 0.2599,E2 249.8851} C_DIS
LIN {X -134.0994,Y -26.5207,Z 192,A -159.4021,B 0.4077,C 0.0713,E1 0.2582,E2 252.7474} C_DIS
LIN {X -134.0994,Y -26.5207,Z 192,A -159.4032,B 0.4077,C 0.0713,E1 0.2582,E2 252.7486} C_DIS
LIN {X -134.8068,Y -22.6407,Z 192,A -161.7092,B 0.4087,C 0.0656,E1 0.2571,E2 255.144} C_DIS
LIN {X -135.2888,Y -19.5566,Z 192,A -163.745,B 0.4095,C 0.0605,E1 0.2562,E2 257.2787} C_DIS
LIN {X -135.7731,Y -15.8514,Z 192,A -166.2546,B 0.4104,C 0.0543,E1 0.2553,E2 259.9152} C_DIS
LIN {X -136.1903,Y -11.7366,Z 192,A -168.8161,B 0.4112,C 0.0477,E1 0.2546,E2 262.5862} C_DIS
LIN {X -136.4452,Y -8.26,Z 192,A -171.1308,B 0.4118,C 0.0418,E1 0.2541,E2 265.0125} C_DIS
LIN {X -136.6356,Y -4.0368,Z 192,A -173.9579,B 0.4125,C 0.0346,E1 0.2538,E2 267.9754} C_DIS
LIN {X -136.6356,Y -4.0368,Z 192,A -173.9589,B 0.4125,C 0.0346,E1 0.2538,E2 267.9765} C_DIS
LIN {X -136.698,Y 0.1044,Z 192,A -176.8199,B 0.413,C 0.0272,E1 0.2538,E2 270.9797} C_DIS
LIN {X -136.698,Y 0.1044,Z 192,A -176.8215,B 0.413,C 0.0272,E1 0.2538,E2 270.9815} C_DIS
LIN {X -136.6305,Y 4.2182,Z 192,A -179.4176,B 0.4134,C 0.0205,E1 0.2539,E2 273.6855} C_DIS
LIN {X -136.6305,Y 4.2182,Z 192,A -179.4186,B 0.4134,C 0.0205,E1 0.2539,E2 273.6866} C_DIS
LIN {X -136.4431,Y 8.2936,Z 192,A 178.0681,B 0.4137,C 0.0139,E1 0.2543,E2 276.2977} C_DIS
LIN {X -136.1497,Y 12.2176,Z 192,A 175.3187,B 0.4139,C 0.0069,E1 0.255,E2 279.179} C_DIS
LIN {X -136.1497,Y 12.2176,Z 192,A 175.3174,B 0.4139,C 0.0069,E1 0.255,E2 279.1805} C_DIS
LIN {X -135.7596,Y 15.9641,Z 192,A 173.1208,B 0.4139,C 0.0011,E1 0.2557,E2 281.4496} C_DIS
LIN {X -135.3333,Y 19.245,Z 192,A 170.9944,B 0.4139,C -0.0043,E1 0.2565,E2 283.6617} C_DIS
LIN {X -134.8512,Y 22.3749,Z 192,A 168.9492,B 0.4139,C -0.0095,E1 0.2575,E2 285.7889} C_DIS
LIN {X -134.2998,Y 25.4766,Z 192,A 166.919,B 0.4137,C -0.0146,E1 0.2585,E2 287.8989} C_DIS
LIN {X -133.6334,Y 28.7675,Z 192,A 164.1763,B 0.4134,C -0.0211,E1 0.2602,E2 290.7889} C_DIS
LIN {X -132.8364,Y 32.2487,Z 192,A 162.4139,B 0.4131,C -0.0257,E1 0.2614,E2 292.5794} C_DIS
LIN {X -131.7618,Y 36.3929,Z 192,A 159.7977,B 0.4127,C -0.032,E1 0.2634,E2 295.283} C_DIS
LIN {X -130.9404,Y 39.2504,Z 192,A 157.8942,B 0.4123,C -0.0365,E1 0.2649,E2 297.2552} C_DIS
LIN {X -129.818,Y 42.8115,Z 192,A 155.557,B 0.4118,C -0.0419,E1 0.267,E2 299.6716} C_DIS
LIN {X -128.6447,Y 46.2165,Z 192,A 153.3776,B 0.4113,C -0.0469,E1 0.2692,E2 301.9182} C_DIS
LIN {X -127.5449,Y 49.1714,Z 192,A 151.4577,B 0.4107,C -0.0512,E1 0.2712,E2 303.8973} C_DIS
LIN {X -126.2143,Y 52.4915,Z 192,A 149.2115,B 0.4101,C -0.0561,E1 0.2737,E2 306.2161} C_DIS
LIN {X -124.8141,Y 55.7387,Z 192,A 147.2674,B 0.4095,C -0.0603,E1 0.276,E2 308.2041} C_DIS
LIN {X -123.476,Y 58.6442,Z 192,A 145.4281,B 0.4089,C -0.0641,E1 0.2783,E2 310.0902} C_DIS
LIN {X -121.9284,Y 61.7971,Z 192,A 143.2909,B 0.4082,C -0.0684,E1 0.2811,E2 312.2889} C_DIS
LIN {X -119.474,Y 66.4224,Z 192,A 140.4429,B 0.4073,C -0.0739,E1 0.2851,E2 315.196} C_DIS
LIN {X -118.1607,Y 68.7316,Z 192,A 138.4016,B 0.4066,C -0.0776,E1 0.2882,E2 317.32} C_DIS
LIN {X -115.4228,Y 73.2365,Z 192,A 135.6118,B 0.4056,C -0.0826,E1 0.2925,E2 320.1595} C_DIS
LIN {X -112.9887,Y 76.939,Z 192,A 133.2036,B 0.4048,C -0.0866,E1 0.2965,E2 322.6142} C_DIS
LIN {X -110.518,Y 80.4472,Z 192,A 131.0775,B 0.404,C -0.0901,E1 0.3002,E2 324.7672} C_DIS
LIN {X -108.2906,Y 83.4217,Z 192,A 128.8704,B 0.4033,C -0.0934,E1 0.3042,E2 327.0278} C_DIS
LIN {X -106.3708,Y 85.8555,Z 192,A 126.5316,B 0.4025,C -0.0964,E1 0.3088,E2 329.4502} C_DIS
LIN {X -103.0296,Y 89.8376,Z 192,A 124.3315,B 0.4018,C -0.0996,E1 0.313,E2 331.6509} C_DIS
LIN {X -98.2071,Y 95.0856,Z 192,A 121.2305,B 0.4008,C -0.1036,E1 0.3193,E2 334.7596} C_DIS
LIN {X -92.8468,Y 100.327,Z 192,A 117.5252,B 0.3997,C -0.1075,E1 0.3274,E2 338.5077} C_DIS
LIN {X -92.8468,Y 100.327,Z 192,A 117.5235,B 0.3997,C -0.1075,E1 0.3274,E2 338.5095} C_DIS
LIN {X -88.5943,Y 104.1007,Z 192,A 114.4975,B 0.399,C -0.1102,E1 0.3343,E2 341.5837} C_DIS
LIN {X -88.5943,Y 104.1007,Z 192,A 114.4964,B 0.399,C -0.1102,E1 0.3343,E2 341.5849} C_DIS
LIN {X -86.0414,Y 106.2209,Z 192,A 112.518,B 0.3986,C -0.1117,E1 0.339,E2 343.6068} C_DIS
LIN {X -82.9314,Y 108.6657,Z 192,A 110.8394,B 0.3982,C -0.113,E1 0.343,E2 345.286} C_DIS
LIN {X -80.3572,Y 110.5832,Z 192,A 109.5541,B 0.3979,C -0.1139,E1 0.3461,E2 346.5663} C_DIS
LIN {X -76.7247,Y 113.1337,Z 192,A 107.514,B 0.3976,C -0.1151,E1 0.3512,E2 348.6188} C_DIS
LIN {X -70.8858,Y 116.8809,Z 192,A 104.4147,B 0.3972,C -0.1166,E1 0.3592,E2 351.7308} C_DIS
LIN {X -68.029,Y 118.5668,Z 192,A 102.7421,B 0.397,C -0.1171,E1 0.3636,E2 353.4233} C_DIS
LIN {X -63.6018,Y 120.9965,Z 192,A 100.8538,B 0.3968,C -0.1177,E1 0.3686,E2 355.294} C_DIS
LIN {X -60.6242,Y 122.5157,Z 192,A 99.4072,B 0.3968,C -0.118,E1 0.3725,E2 356.7433} C_DIS
LIN {X -57.1434,Y 124.1775,Z 192,A 97.4782,B 0.3968,C -0.118,E1 0.3779,E2 358.6942} C_DIS
LIN {X -51.7294,Y 126.5302,Z 192,A 95.1882,B 0.3967,C -0.1182,E1 0.3842,E2 360.9698} C_DIS
LIN {X -46.5418,Y 128.5272,Z 192,A 92.3425,B 0.3969,C -0.1176,E1 0.3924,E2 363.8515} C_DIS
LIN {X -41.7549,Y 130.1613,Z 192,A 90.8897,B 0.3969,C -0.1176,E1 0.3964,E2 365.2554} C_DIS
LIN {X -38.4082,Y 131.1877,Z 192,A 89.4535,B 0.3969,C -0.1172,E1 0.4006,E2 366.6886} C_DIS
LIN {X -34.2264,Y 132.3418,Z 192,A 87.7351,B 0.3972,C -0.1166,E1 0.4056,E2 368.3991} C_DIS
LIN {X -30.6123,Y 133.2229,Z 192,A 86.2723,B 0.3973,C -0.116,E1 0.4098,E2 369.854} C_DIS
LIN {X -27.1859,Y 133.9641,Z 192,A 84.9393,B 0.3975,C -0.1154,E1 0.4137,E2 371.1764} C_DIS
LIN {X -22.999,Y 134.747,Z 192,A 82.6843,B 0.398,C -0.1137,E1 0.4206,E2 373.4652} C_DIS
LIN {X -18.0452,Y 135.4988,Z 192,A 81.2554,B 0.3982,C -0.1131,E1 0.4247,E2 374.8437} C_DIS
LIN {X -12.9038,Y 136.0845,Z 192,A 79.5136,B 0.3985,C -0.112,E1 0.4298,E2 376.5526} C_DIS
LIN {X -4.5006,Y 136.6227,Z 192,A 75.3023,B 0.3997,C -0.1077,E1 0.4426,E2 380.8138} C_DIS
LIN {X 2.6397,Y 136.67,Z 192,A 73.8077,B 0.3999,C -0.107,E1 0.4467,E2 382.1934} C_DIS
LIN {X 2.6397,Y 136.67,Z 192,A 73.8065,B 0.3999,C -0.107,E1 0.4467,E2 382.1947} C_DIS
LIN {X 9.6004,Y 136.3578,Z 192,A 71.2311,B 0.4006,C -0.1043,E1 0.4543,E2 384.7422} C_DIS
LIN {X 9.6004,Y 136.3578,Z 192,A 71.2297,B 0.4006,C -0.1043,E1 0.4543,E2 384.7436} C_DIS
LIN {X 14.7238,Y 135.8996,Z 192,A 69.1758,B 0.4012,C -0.1018,E1 0.4604,E2 386.7888} C_DIS
LIN {X 18.5506,Y 135.4323,Z 192,A 67.6788,B 0.4017,C -0.0999,E1 0.4647,E2 388.2759} C_DIS
LIN {X 23.4746,Y 134.6654,Z 192,A 65.9755,B 0.4022,C -0.0977,E1 0.4696,E2 389.9476} C_DIS
LIN {X 27.4944,Y 133.9013,Z 192,A 64.5549,B 0.4027,C -0.0959,E1 0.4737,E2 391.3436} C_DIS
LIN {X 31.727,Y 132.9621,Z 192,A 63.1351,B 0.4031,C -0.094,E1 0.4777,E2 392.7302} C_DIS
LIN {X 35.1668,Y 132.0936,Z 192,A 61.8715,B 0.4035,C -0.0921,E1 0.4812,E2 393.9749} C_DIS
LIN {X 38.5864,Y 131.1356,Z 192,A 60.6267,B 0.404,C -0.0903,E1 0.4847,E2 395.1988} C_DIS
LIN {X 42.3197,Y 129.9808,Z 192,A 59.154,B 0.4045,C -0.0879,E1 0.4888,E2 396.6572} C_DIS
LIN {X 45.372,Y 128.9464,Z 192,A 57.5019,B 0.4051,C -0.0848,E1 0.4935,E2 398.3346} C_DIS
LIN {X 51.0636,Y 126.7986,Z 192,A 56.1466,B 0.4055,C -0.0833,E1 0.4969,E2 399.587} C_DIS
LIN {X 55.876,Y 124.7527,Z 192,A 54.3263,B 0.4061,C -0.0802,E1 0.5016,E2 401.3744} C_DIS
LIN {X 59.1103,Y 123.2533,Z 192,A 53.1112,B 0.4065,C -0.0781,E1 0.5048,E2 402.5644} C_DIS
LIN {X 62.6103,Y 121.5144,Z 192,A 51.7087,B 0.407,C -0.0756,E1 0.5084,E2 403.9457} C_DIS
LIN {X 65.7813,Y 119.8285,Z 192,A 50.0478,B 0.4076,C -0.0721,E1 0.5126,E2 405.6204} C_DIS
LIN {X 70.5599,Y 117.078,Z 192,A 48.6986,B 0.4079,C -0.0701,E1 0.5158,E2 406.8821} C_DIS
LIN {X 73.3951,Y 115.3221,Z 192,A 47.4344,B 0.4084,C -0.0676,E1 0.5188,E2 408.1338} C_DIS
LIN {X 76.1776,Y 113.5033,Z 192,A 46.4989,B 0.4086,C -0.066,E1 0.521,E2 409.0266} C_DIS
LIN {X 79.878,Y 110.9306,Z 192,A 45.0326,B 0.4091,C -0.0631,E1 0.5243,E2 410.4529} C_DIS
LIN {X 83.391,Y 108.3145,Z 192,A 43.5436,B 0.4095,C -0.0602,E1 0.5277,E2 411.9087} C_DIS
LIN {X 86.9829,Y 105.4512,Z 192,A 42.0587,B 0.41,C -0.0572,E1 0.5309,E2 413.3511} C_DIS
LIN {X 90.3224,Y 102.6053,Z 192,A 40.6336,B 0.4103,C -0.0543,E1 0.5339,E2 414.7357} C_DIS
LIN {X 93.4681,Y 99.7487,Z 192,A 39.2509,B 0.4107,C -0.0514,E1 0.5367,E2 416.079} C_DIS
LIN {X 96.6629,Y 96.656,Z 192,A 37.7881,B 0.4111,C -0.0484,E1 0.5396,E2 417.5018} C_DIS
LIN {X 99.8273,Y 93.3837,Z 192,A 36.3259,B 0.4114,C -0.0453,E1 0.5424,E2 418.919} C_DIS
LIN {X 102.8083,Y 90.0913,Z 192,A 34.8952,B 0.4118,C -0.0422,E1 0.545,E2 420.3058} C_DIS
LIN {X 105.5972,Y 86.8061,Z 192,A 33.5121,B 0.4121,C -0.0392,E1 0.5475,E2 421.6454} C_DIS
LIN {X 108.3068,Y 83.401,Z 192,A 32.1019,B 0.4123,C -0.0361,E1 0.5499,E2 423.0125} C_DIS
LIN {X 110.8802,Y 79.9475,Z 192,A 30.7468,B 0.4126,C -0.0331,E1 0.5521,E2 424.3203} C_DIS
LIN {X 115.4404,Y 73.2086,Z 192,A 28.1208,B 0.413,C -0.0272,E1 0.556,E2 426.8625} C_DIS
LIN {X 118.884,Y 67.4729,Z 192,A 26.0118,B 0.4133,C -0.0224,E1 0.559,E2 428.8961} C_DIS
LIN {X 120.8565,Y 63.8684,Z 192,A 24.756,B 0.4135,C -0.0196,E1 0.5606,E2 430.1006} C_DIS
LIN {X 122.3369,Y 60.9866,Z 192,A 23.7461,B 0.4135,C -0.0173,E1 0.5618,E2 431.0719} C_DIS
LIN {X 123.5395,Y 58.5112,Z 192,A 22.3506,B 0.4137,C -0.0133,E1 0.5635,E2 432.4948} C_DIS
LIN {X 125.8236,Y 53.427,Z 192,A 21.116,B 0.4137,C -0.0112,E1 0.5648,E2 433.6056} C_DIS
LIN {X 128.7431,Y 45.9435,Z 192,A 18.4707,B 0.4139,C -0.0049,E1 0.5673,E2 436.1685} C_DIS
LIN {X 130.1351,Y 41.8367,Z 192,A 17.1989,B 0.4139,C -0.002,E1 0.5684,E2 437.3771} C_DIS
LIN {X 131.1077,Y 38.6815,Z 192,A 16.1559,B 0.4139,C 0.0004,E1 0.5692,E2 438.3803} C_DIS
LIN {X 132.0792,Y 35.2207,Z 192,A 15.0152,B 0.4139,C 0.0031,E1 0.57,E2 439.4779} C_DIS
LIN {X 132.8643,Y 32.1329,Z 192,A 14.0237,B 0.4139,C 0.0055,E1 0.5706,E2 440.4287} C_DIS
LIN {X 133.5758,Y 29.034,Z 192,A 13.0141,B 0.4139,C 0.0079,E1 0.5712,E2 441.3999} C_DIS
LIN {X 134.228,Y 25.852,Z 192,A 11.9497,B 0.4138,C 0.0105,E1 0.5718,E2 442.4288} C_DIS
LIN {X 135.0034,Y 21.4437,Z 192,A 10.5164,B 0.4137,C 0.0139,E1 0.5724,E2 443.8086} C_DIS
LIN {X 135.463,Y 18.3179,Z 192,A 9.0471,B 0.4135,C 0.0182,E1 0.573,E2 445.2964} C_DIS
LIN {X 136.0937,Y 12.8083,Z 192,A 7.9119,B 0.4135,C 0.0199,E1 0.5733,E2 446.2853} C_DIS
LIN {X 136.5837,Y 5.5161,Z 192,A 5.6973,B 0.4132,C 0.025,E1 0.5737,E2 448.3943} C_DIS
LIN {X 136.5837,Y 5.5161,Z 192,A 5.6962,B 0.4132,C 0.025,E1 0.5737,E2 448.3955} C_DIS
LIN {X 136.6903,Y 1.2842,Z 192,A 3.896,B 0.4128,C 0.03,E1 0.5737,E2 450.2} C_DIS
LIN {X 136.6728,Y -2.4704,Z 192,A 2.4209,B 0.4125,C 0.034,E1 0.5737,E2 451.6633} C_DIS
LIN {X 136.4325,Y -8.4669,Z 192,A 1.0762,B 0.4123,C 0.0363,E1 0.5735,E2 452.8586} C_DIS
LIN {X 135.6073,Y -17.2176,Z 192,A -1.7754,B 0.4117,C 0.0431,E1 0.5727,E2 455.6032} C_DIS
LIN {X 134.9813,Y -21.5866,Z 192,A -3.147,B 0.4113,C 0.0463,E1 0.5721,E2 456.9126} C_DIS
LIN {X 134.3052,Y -25.4483,Z 192,A -4.32,B 0.411,C 0.0489,E1 0.5716,E2 458.0238} C_DIS
LIN {X 133.6247,Y -28.8075,Z 192,A -5.4305,B 0.4107,C 0.0515,E1 0.571,E2 459.0913} C_DIS
LIN {X 132.6255,Y -33.1086,Z 192,A -6.846,B 0.4103,C 0.0548,E1 0.5701,E2 460.4492} C_DIS
LIN {X 131.6914,Y -36.6445,Z 192,A -7.9276,B 0.41,C 0.0572,E1 0.5693,E2 461.4704} C_DIS
LIN {X 130.5606,Y -40.4917,Z 192,A -9.9186,B 0.4091,C 0.063,E1 0.5676,E2 463.5048} C_DIS
LIN {X 128.3448,Y -47.0481,Z 192,A -11.4938,B 0.4087,C 0.0655,E1 0.5663,E2 464.9} C_DIS
LIN {X 127.0461,Y -50.4497,Z 192,A -12.9918,B 0.4081,C 0.0694,E1 0.5648,E2 466.3952} C_DIS
LIN {X 125.2402,Y -54.7777,Z 192,A -14.187,B 0.4077,C 0.0716,E1 0.5636,E2 467.4844} C_DIS
LIN {X 123.5393,Y -58.5116,Z 192,A -15.419,B 0.4072,C 0.0741,E1 0.5622,E2 468.649} C_DIS
LIN {X 122.002,Y -61.6525,Z 192,A -16.4944,B 0.4068,C 0.0764,E1 0.5609,E2 469.6703} C_DIS
LIN {X 120.058,Y -65.3606,Z 192,A -17.934,B 0.4062,C 0.0797,E1 0.5591,E2 471.0663} C_DIS
LIN {X 117.8664,Y -69.2346,Z 192,A -19.5872,B 0.4054,C 0.0837,E1 0.5568,E2 472.6907} C_DIS
LIN {X 115.8039,Y -72.6329,Z 192,A -20.6558,B 0.405,C 0.0856,E1 0.5553,E2 473.6749} C_DIS
LIN {X 112.8513,Y -77.1388,Z 192,A -22.4379,B 0.4041,C 0.0895,E1 0.5526,E2 475.39} C_DIS
LIN {X 110.3511,Y -80.6755,Z 192,A -24.1738,B 0.4032,C 0.0937,E1 0.5497,E2 477.1158} C_DIS
LIN {X 107.2042,Y -84.8135,Z 192,A -25.4819,B 0.4027,C 0.0957,E1 0.5477,E2 478.2988} C_DIS
LIN {X 104.361,Y -88.2881,Z 192,A -26.931,B 0.402,C 0.0986,E1 0.5451,E2 479.6859} C_DIS
LIN {X 100.3404,Y -92.8317,Z 192,A -29.0659,B 0.4009,C 0.1031,E1 0.5412,E2 481.7626} C_DIS
LIN {X 97.9615,Y -95.3393,Z 192,A -30.0377,B 0.4005,C 0.1047,E1 0.5394,E2 482.6649} C_DIS
LIN {X 94.8404,Y -98.4445,Z 192,A -31.4787,B 0.3997,C 0.1075,E1 0.5365,E2 484.0471} C_DIS
LIN {X 91.8393,Y -101.2494,Z 192,A -32.899,B 0.3989,C 0.1103,E1 0.5336,E2 485.4238} C_DIS
LIN {X 86.9552,Y -105.4741,Z 192,A -34.9687,B 0.3979,C 0.1141,E1 0.5293,E2 487.3999} C_DIS
LIN {X 83.4567,Y -108.2636,Z 192,A -36.4672,B 0.3971,C 0.1168,E1 0.5261,E2 488.8431} C_DIS
LIN {X 80.3565,Y -110.5838,Z 192,A -37.7504,B 0.3964,C 0.1191,E1 0.5232,E2 490.0762} C_DIS
LIN {X 75.5984,Y -113.8899,Z 192,A -39.685,B 0.3954,C 0.1225,E1 0.5188,E2 491.9376} C_DIS
LIN {X 71.2075,Y -116.6851,Z 192,A -41.7772,B 0.3941,C 0.1266,E1 0.5136,E2 494.018} C_DIS
LIN {X 67.1628,Y -119.0593,Z 192,A -43.0282,B 0.3936,C 0.1281,E1 0.5108,E2 495.1612} C_DIS
LIN {X 63.4321,Y -121.0857,Z 192,A -44.3674,B 0.3929,C 0.1301,E1 0.5075,E2 496.4341} C_DIS
LIN {X 60.7422,Y -122.4574,Z 192,A -45.4111,B 0.3924,C 0.1318,E1 0.5049,E2 497.4445} C_DIS
LIN {X 58.0687,Y -123.7496,Z 192,A -46.5142,B 0.3918,C 0.1336,E1 0.502,E2 498.5269} C_DIS
LIN {X 52.5606,Y -126.1855,Z 192,A -48.8165,B 0.3904,C 0.1375,E1 0.4959,E2 500.7968} C_DIS
LIN {X 48.7328,Y -127.7153,Z 192,A -49.9744,B 0.39,C 0.1387,E1 0.493,E2 501.8677} C_DIS
LIN {X 45.2156,Y -129.0006,Z 192,A -51.4163,B 0.3892,C 0.141,E1 0.4891,E2 503.2909} C_DIS
LIN {X 40.3749,Y -130.5964,Z 192,A -53.0321,B 0.3885,C 0.1429,E1 0.4848,E2 504.8271} C_DIS
LIN {X 36.9592,Y -131.6034,Z 192,A -54.2249,B 0.3879,C 0.1444,E1 0.4815,E2 505.9742} C_DIS
LIN {X 33.878,Y -132.4302,Z 192,A -55.3839,B 0.3873,C 0.146,E1 0.4783,E2 507.1063} C_DIS
LIN {X 30.4935,Y -133.2501,Z 192,A -56.6474,B 0.3867,C 0.1476,E1 0.4747,E2 508.3401} C_DIS
LIN {X 26.0379,Y -134.1925,Z 192,A -58.216,B 0.386,C 0.1494,E1 0.4703,E2 509.8566} C_DIS
LIN {X 23.2017,Y -134.7132,Z 192,A -60.0527,B 0.3847,C 0.1527,E1 0.4647,E2 511.7933} C_DIS
LIN {X 16.3221,Y -135.7169,Z 192,A -62.5419,B 0.3837,C 0.1553,E1 0.4575,E2 514.2178} C_DIS
LIN {X 9.4858,Y -136.3662,Z 192,A -64.3354,B 0.3834,C 0.156,E1 0.4527,E2 515.8421} C_DIS
LIN {X 6.3136,Y -136.5502,Z 192,A -65.9588,B 0.3825,C 0.1582,E1 0.4477,E2 517.5128} C_DIS
LIN {X 1.2048,Y -136.6904,Z 192,A -67.2932,B 0.3823,C 0.1586,E1 0.4441,E2 518.7206} C_DIS
LIN {X 1.2048,Y -136.6904,Z 192,A -67.2935,B 0.3823,C 0.1586,E1 0.4441,E2 518.721} C_DIS
Enddeposition()
LIN {X 0.9892,Y -137.59,Z 192,A -67.4352,B 0.4038,C 0.1594,E1 0.4652,E2 518.8771} C_DIS
Startdeposition()
$VEL.CP = VEL_PRINT
LIN {X 6.1124,Y -137.4597,Z 192,A -65.65,B 0.4044,C 0.158,E1 0.4703,E2 517.1463} C_DIS
LIN {X 9.8835,Y -137.2384,Z 192,A -64.0473,B 0.4051,C 0.1561,E1 0.4751,E2 515.5377} C_DIS
LIN {X 13.5094,Y -136.9294,Z 192,A -62.7536,B 0.4055,C 0.1549,E1 0.4788,E2 514.2783} C_DIS
LIN {X 16.9599,Y -136.5461,Z 192,A -61.228,B 0.4063,C 0.1529,E1 0.4833,E2 512.7389} C_DIS
LIN {X 22.0186,Y -135.822,Z 192,A -59.9418,B 0.4065,C 0.1524,E1 0.4867,E2 511.5853} C_DIS
LIN {X 24.7672,Y -135.3473,Z 192,A -58.6219,B 0.4072,C 0.1504,E1 0.4906,E2 510.2393} C_DIS
LIN {X 28.3227,Y -134.649,Z 192,A -57.642,B 0.4075,C 0.1497,E1 0.4932,E2 509.3422} C_DIS
LIN {X 30.8502,Y -134.0907,Z 192,A -56.6748,B 0.4079,C 0.1485,E1 0.4959,E2 508.3917} C_DIS
LIN {X 34.6594,Y -133.1592,Z 192,A -55.3035,B 0.4085,C 0.1468,E1 0.4997,E2 507.0606} C_DIS
LIN {X 37.217,Y -132.4647,Z 192,A -54.3609,B 0.409,C 0.1456,E1 0.5023,E2 506.1425} C_DIS
LIN {X 40.6183,Y -131.462,Z 192,A -53.087,B 0.4096,C 0.1439,E1 0.5058,E2 504.8994} C_DIS
LIN {X 44.0659,Y -130.3478,Z 192,A -51.8536,B 0.4102,C 0.1422,E1 0.5091,E2 503.7082} C_DIS
LIN {X 47.5506,Y -129.118,Z 192,A -50.4642,B 0.4109,C 0.1401,E1 0.5129,E2 502.341} C_DIS
LIN {X 55.2383,Y -126.0204,Z 192,A -47.7411,B 0.4121,C 0.1364,E1 0.5199,E2 499.7294} C_DIS
LIN {X 58.5945,Y -124.4959,Z 192,A -46.439,B 0.4128,C 0.1343,E1 0.5232,E2 498.4624} C_DIS
LIN {X 61.4545,Y -123.1084,Z 192,A -45.2915,B 0.4134,C 0.1325,E1 0.5262,E2 497.3412} C_DIS
LIN {X 65.3755,Y -121.0728,Z 192,A -43.3915,B 0.4146,C 0.1287,E1 0.531,E2 495.4303} C_DIS
LIN {X 69.511,Y -118.7466,Z 192,A -42.1573,B 0.415,C 0.1274,E1 0.5339,E2 494.3096} C_DIS
LIN {X 73.1218,Y -116.5583,Z 192,A -40.7321,B 0.4157,C 0.125,E1 0.5372,E2 492.9344} C_DIS
LIN {X 77.6459,Y -113.5942,Z 192,A -38.9019,B 0.4167,C 0.1218,E1 0.5415,E2 491.1675} C_DIS
LIN {X 81.2293,Y -111.0601,Z 192,A -37.4727,B 0.4174,C 0.1194,E1 0.5447,E2 489.7979} C_DIS
LIN {X 84.5245,Y -108.5734,Z 192,A -36.0457,B 0.4181,C 0.1167,E1 0.5478,E2 488.4142} C_DIS
LIN {X 88.0128,Y -105.7655,Z 192,A -34.5277,B 0.4189,C 0.1139,E1 0.5511,E2 486.9474} C_DIS
LIN {X 90.9535,Y -103.2472,Z 192,A -33.2583,B 0.4195,C 0.1115,E1 0.5537,E2 485.7288} C_DIS
LIN {X 94.2532,Y -100.244,Z 192,A -31.7981,B 0.4203,C 0.1088,E1 0.5566,E2 484.3274} C_DIS
LIN {X 97.3262,Y -97.2638,Z 192,A -30.3808,B 0.421,C 0.1061,E1 0.5594,E2 482.9637} C_DIS
LIN {X 100.3868,Y -94.1015,Z 192,A -28.9915,B 0.4216,C 0.1034,E1 0.562,E2 481.6394} C_DIS
LIN {X 102.4075,Y -91.8978,Z 192,A -27.942,B 0.4221,C 0.1012,E1 0.5639,E2 480.6182} C_DIS
LIN {X 105.401,Y -88.4483,Z 192,A -26.4528,B 0.4228,C 0.0983,E1 0.5666,E2 479.189} C_DIS
LIN {X 108.1973,Y -85.0048,Z 192,A -24.9236,B 0.4236,C 0.095,E1 0.5692,E2 477.7055} C_DIS
LIN {X 112.3337,Y -79.4585,Z 192,A -22.363,B 0.4249,C 0.0891,E1 0.5734,E2 475.1901} C_DIS
LIN {X 115.2247,Y -75.2054,Z 192,A -21.2383,B 0.4252,C 0.0877,E1 0.5749,E2 474.2131} C_DIS
LIN {X 118.3036,Y -70.2623,Z 192,A -19.3599,B 0.426,C 0.0838,E1 0.5776,E2 472.4125} C_DIS
LIN {X 118.3036,Y -70.2623,Z 192,A -19.3608,B 0.426,C 0.0838,E1 0.5776,E2 472.4135} C_DIS
LIN {X 119.8459,Y -67.598,Z 192,A -18.2263,B 0.4265,C 0.081,E1 0.5791,E2 471.2995} C_DIS
LIN {X 121.8719,Y -63.8682,Z 192,A -16.9073,B 0.427,C 0.0782,E1 0.5808,E2 470.0438} C_DIS
LIN {X 123.4216,Y -60.8195,Z 192,A -15.7708,B 0.4275,C 0.0757,E1 0.5822,E2 468.9476} C_DIS
LIN {X 125.0257,Y -57.4509,Z 192,A -14.5806,B 0.4279,C 0.0731,E1 0.5835,E2 467.8082} C_DIS
LIN {X 127.0889,Y -52.7299,Z 192,A -12.9509,B 0.4285,C 0.0695,E1 0.5852,E2 466.2503} C_DIS
LIN {X 128.538,Y -49.0976,Z 192,A -11.6015,B 0.429,C 0.0663,E1 0.5866,E2 464.9391} C_DIS
LIN {X 129.936,Y -45.2617,Z 192,A -10.1748,B 0.4295,C 0.0628,E1 0.5879,E2 463.5498} C_DIS
LIN {X 131.0187,Y -42.025,Z 192,A -9.3054,B 0.4298,C 0.0612,E1 0.5886,E2 462.7567} C_DIS
LIN {X 132.0758,Y -38.574,Z 192,A -8.1646,B 0.4301,C 0.0587,E1 0.5894,E2 461.6651} C_DIS
LIN {X 132.9835,Y -35.3183,Z 192,A -7.0682,B 0.4305,C 0.0561,E1 0.5902,E2 460.6109} C_DIS
LIN {X 133.7759,Y -32.1868,Z 192,A -6.0447,B 0.4308,C 0.0537,E1 0.5909,E2 459.6308} C_DIS
LIN {X 134.6536,Y -28.3014,Z 192,A -4.7665,B 0.4311,C 0.0508,E1 0.5916,E2 458.4037} C_DIS
LIN {X 135.3801,Y -24.5838,Z 192,A -3.5534,B 0.4315,C 0.0479,E1 0.5922,E2 457.2392} C_DIS
LIN {X 135.987,Y -20.9655,Z 192,A -2.1396,B 0.4319,C 0.0442,E1 0.5928,E2 455.8399} C_DIS
LIN {X 136.5323,Y -17.0761,Z 192,A -1.1865,B 0.432,C 0.0425,E1 0.5931,E2 454.9779} C_DIS
LIN {X 136.9475,Y -13.3215,Z 192,A 0.054,B 0.4323,C 0.0395,E1 0.5935,E2 453.7809} C_DIS
LIN {X 137.256,Y -9.6431,Z 192,A 1.2381,B 0.4326,C 0.0367,E1 0.5937,E2 452.643} C_DIS
LIN {X 137.4425,Y -6.467,Z 192,A 2.4768,B 0.4328,C 0.0333,E1 0.5939,E2 451.4149} C_DIS
LIN {X 137.5668,Y -2.7722,Z 192,A 3.3244,B 0.4329,C 0.0319,E1 0.5939,E2 450.6576} C_DIS
LIN {X 137.5701,Y 2.5738,Z 192,A 5.0405,B 0.4332,C 0.0278,E1 0.5939,E2 449.0068} C_DIS
LIN {X 137.467,Y 5.9346,Z 192,A 6.5474,B 0.4335,C 0.0235,E1 0.5937,E2 447.4853} C_DIS
LIN {X 137.1837,Y 10.6333,Z 192,A 7.7078,B 0.4335,C 0.0213,E1 0.5935,E2 446.4272} C_DIS
LIN {X 136.5687,Y 16.7708,Z 192,A 9.6968,B 0.4338,C 0.0165,E1 0.5929,E2 444.5108} C_DIS
LIN {X 136.0526,Y 20.5422,Z 192,A 11.1218,B 0.4339,C 0.0127,E1 0.5923,E2 443.1055} C_DIS
LIN {X 135.3881,Y 24.5392,Z 192,A 12.0415,B 0.4339,C 0.0112,E1 0.592,E2 442.2813} C_DIS
LIN {X 134.8206,Y 27.4845,Z 192,A 13.0179,B 0.434,C 0.0088,E1 0.5914,E2 441.3382} C_DIS
LIN {X 134.0826,Y 30.8855,Z 192,A 14.1497,B 0.434,C 0.0061,E1 0.5908,E2 440.245} C_DIS
LIN {X 133.0554,Y 35.0488,Z 192,A 15.542,B 0.4341,C 0.0028,E1 0.5898,E2 438.9002} C_DIS
LIN {X 131.9478,Y 39.0113,Z 192,A 16.793,B 0.4341,C -0.0001,E1 0.5889,E2 437.7049} C_DIS
LIN {X 130.94,Y 42.2712,Z 192,A 17.8836,B 0.4341,C -0.0027,E1 0.588,E2 436.6536} C_DIS
LIN {X 129.7371,Y 45.8356,Z 192,A 19.3613,B 0.4341,C -0.0066,E1 0.5867,E2 435.186} C_DIS
LIN {X 128.4774,Y 49.2535,Z 192,A 20.1895,B 0.4341,C -0.008,E1 0.5859,E2 434.4393} C_DIS
LIN {X 126.8704,Y 53.2532,Z 192,A 21.6697,B 0.434,C -0.0116,E1 0.5844,E2 432.9957} C_DIS
LIN {X 124.5754,Y 58.4246,Z 192,A 23.4202,B 0.4338,C -0.0156,E1 0.5824,E2 431.3152} C_DIS
LIN {X 123.2177,Y 61.233,Z 192,A 24.4476,B 0.4338,C -0.018,E1 0.5812,E2 430.3188} C_DIS
LIN {X 121.0869,Y 65.3491,Z 192,A 25.9729,B 0.4336,C -0.0215,E1 0.5793,E2 428.8395} C_DIS
LIN {X 118.844,Y 69.3451,Z 192,A 27.4448,B 0.4334,C -0.0249,E1 0.5773,E2 427.4167} C_DIS
LIN {X 116.555,Y 73.1269,Z 192,A 28.8758,B 0.4332,C -0.0281,E1 0.5752,E2 426.0315} C_DIS
LIN {X 113.6895,Y 77.5071,Z 192,A 30.4357,B 0.433,C -0.0314,E1 0.5729,E2 424.54} C_DIS
LIN {X 111.6399,Y 80.4311,Z 192,A 31.7235,B 0.4327,C -0.0345,E1 0.5708,E2 423.2739} C_DIS
LIN {X 108.958,Y 84.0282,Z 192,A 33.146,B 0.4325,C -0.0375,E1 0.5684,E2 421.8998} C_DIS
LIN {X 106.2348,Y 87.446,Z 192,A 34.5808,B 0.4322,C -0.0407,E1 0.566,E2 420.5064} C_DIS
LIN {X 103.278,Y 90.9187,Z 192,A 36.0495,B 0.4319,C -0.0438,E1 0.5633,E2 419.0836} C_DIS
LIN {X 100.2401,Y 94.2573,Z 192,A 37.5214,B 0.4316,C -0.0469,E1 0.5605,E2 417.6547} C_DIS
LIN {X 97.0409,Y 97.5477,Z 192,A 39.0013,B 0.4312,C -0.05,E1 0.5577,E2 416.2199} C_DIS
LIN {X 93.8154,Y 100.6536,Z 192,A 40.4687,B 0.4309,C -0.053,E1 0.5547,E2 414.7935} C_DIS
LIN {X 90.6142,Y 103.545,Z 192,A 41.8932,B 0.4305,C -0.0559,E1 0.5517,E2 413.4071} C_DIS
LIN {X 87.0459,Y 106.5621,Z 192,A 43.4121,B 0.4301,C -0.0589,E1 0.5485,E2 411.9315} C_DIS
LIN {X 83.3912,Y 109.4461,Z 192,A 44.9568,B 0.4297,C -0.062,E1 0.5451,E2 410.4264} C_DIS
LIN {X 79.6718,Y 112.1832,Z 192,A 46.4989,B 0.4292,C -0.0649,E1 0.5416,E2 408.9221} C_DIS
LIN {X 75.8851,Y 114.778,Z 192,A 47.9838,B 0.4288,C -0.0677,E1 0.5381,E2 407.4792} C_DIS
LIN {X 72.2746,Y 117.0855,Z 192,A 49.4732,B 0.4283,C -0.0705,E1 0.5345,E2 406.0186} C_DIS
LIN {X 67.5485,Y 119.8737,Z 192,A 51.2853,B 0.4278,C -0.0737,E1 0.5301,E2 404.2521} C_DIS
LIN {X 63.5906,Y 122.0177,Z 192,A 52.7126,B 0.4274,C -0.0762,E1 0.5266,E2 402.8673} C_DIS
LIN {X 60.1698,Y 123.7422,Z 192,A 54.0194,B 0.427,C -0.0784,E1 0.5233,E2 401.5877} C_DIS
LIN {X 57.2958,Y 125.0974,Z 192,A 55.1957,B 0.4266,C -0.0805,E1 0.5202,E2 400.4252} C_DIS
LIN {X 54.1214,Y 126.5033,Z 192,A 56.3136,B 0.4263,C -0.0822,E1 0.5173,E2 399.3378} C_DIS
LIN {X 50.2167,Y 128.103,Z 192,A 57.91,B 0.4257,C -0.085,E1 0.513,E2 397.7565} C_DIS
LIN {X 44.7485,Y 130.114,Z 192,A 59.7574,B 0.4252,C -0.0876,E1 0.5081,E2 395.962} C_DIS
LIN {X 41.794,Y 131.0924,Z 192,A 60.8085,B 0.4249,C -0.0892,E1 0.5052,E2 394.933} C_DIS
LIN {X 37.9706,Y 132.2525,Z 192,A 62.3058,B 0.4244,C -0.0915,E1 0.501,E2 393.451} C_DIS
LIN {X 34.0428,Y 133.3158,Z 192,A 63.6244,B 0.424,C -0.0932,E1 0.4974,E2 392.1658} C_DIS
LIN {X 30.7652,Y 134.1101,Z 192,A 64.809,B 0.4236,C -0.0948,E1 0.494,E2 391.0008} C_DIS
LIN {X 27.0304,Y 134.9131,Z 192,A 66.1772,B 0.4232,C -0.0966,E1 0.4901,E2 389.6522} C_DIS
LIN {X 23.5811,Y 135.5595,Z 192,A 68.0092,B 0.4226,C -0.0994,E1 0.4847,E2 387.7887} C_DIS
LIN {X 18.3094,Y 136.3708,Z 192,A 69.1876,B 0.4224,C -0.1002,E1 0.4816,E2 386.7003} C_DIS
LIN {X 12.7137,Y 137.0058,Z 192,A 71.4243,B 0.4217,C -0.1029,E1 0.475,E2 384.4735} C_DIS
LIN {X 8.7479,Y 137.3158,Z 192,A 72.8374,B 0.4214,C -0.1044,E1 0.4709,E2 383.0813} C_DIS
LIN {X 5.0855,Y 137.5001,Z 192,A 74.2114,B 0.421,C -0.1058,E1 0.4668,E2 381.7204} C_DIS
LIN {X -1.5504,Y 137.5872,Z 192,A 76.5666,B 0.4205,C -0.1079,E1 0.4599,E2 379.4} C_DIS
LIN {X -4.359,Y 137.5259,Z 192,A 78.1692,B 0.42,C -0.1096,E1 0.455,E2 377.7622} C_DIS
LIN {X -9.0878,Y 137.2948,Z 192,A 79.4015,B 0.42,C -0.1102,E1 0.4516,E2 376.5911} C_DIS
LIN {X -12.815,Y 136.9961,Z 192,A 80.8995,B 0.4196,C -0.1113,E1 0.4471,E2 375.0983} C_DIS
LIN {X -16.2729,Y 136.6281,Z 192,A 82.5326,B 0.4193,C -0.1126,E1 0.4422,E2 373.4508} C_DIS
LIN {X -20.0455,Y 136.127,Z 192,A 83.804,B 0.4191,C -0.1132,E1 0.4385,E2 372.2054} C_DIS
LIN {X -24.2507,Y 135.4397,Z 192,A 85.2887,B 0.4189,C -0.1139,E1 0.4342,E2 370.7445} C_DIS
LIN {X -27.5442,Y 134.8085,Z 192,A 86.6054,B 0.4187,C -0.1145,E1 0.4304,E2 369.4346} C_DIS
LIN {X -30.9335,Y 134.0716,Z 192,A 88.0362,B 0.4186,C -0.1151,E1 0.4262,E2 368.0055} C_DIS
LIN {X -35.1577,Y 133.0264,Z 192,A 89.7613,B 0.4184,C -0.1157,E1 0.4212,E2 366.288} C_DIS
LIN {X -38.7703,Y 132.0183,Z 192,A 91.2228,B 0.4184,C -0.116,E1 0.417,E2 364.8351} C_DIS
LIN {X -41.8779,Y 131.0656,Z 192,A 93.4659,B 0.4181,C -0.1169,E1 0.4104,E2 362.5216} C_DIS
LIN {X -48.1109,Y 128.9081,Z 192,A 94.9868,B 0.4182,C -0.1164,E1 0.4064,E2 361.0992} C_DIS
LIN {X -48.1109,Y 128.9081,Z 192,A 94.9858,B 0.4182,C -0.1164,E1 0.4064,E2 361.1003} C_DIS
LIN {X -51.9571,Y 127.4077,Z 192,A 97.5409,B 0.4182,C -0.1168,E1 0.3991,E2 358.4803} C_DIS
LIN {X -56.1507,Y 125.6146,Z 192,A 98.5729,B 0.4182,C -0.1162,E1 0.3964,E2 357.5173} C_DIS
LIN {X -56.1507,Y 125.6146,Z 192,A 98.5719,B 0.4182,C -0.1162,E1 0.3964,E2 357.5185} C_DIS
LIN {X -59.5343,Y 124.047,Z 192,A 100.5227,B 0.4183,C -0.1161,E1 0.391,E2 355.5373} C_DIS
LIN {X -63.1167,Y 122.2653,Z 192,A 102.3437,B 0.4184,C -0.1157,E1 0.3861,E2 353.705} C_DIS
LIN {X -67.3011,Y 120.0127,Z 192,A 104.3432,B 0.4186,C -0.1149,E1 0.3809,E2 351.7048} C_DIS
LIN {X -70.8559,Y 117.9495,Z 192,A 106.1779,B 0.4188,C -0.1142,E1 0.3761,E2 349.8611} C_DIS
LIN {X -74.7624,Y 115.5123,Z 192,A 108.2357,B 0.4191,C -0.1131,E1 0.3709,E2 347.7931} C_DIS
LIN {X -78.2727,Y 113.1636,Z 192,A 110.7819,B 0.4195,C -0.1118,E1 0.3645,E2 345.1841} C_DIS
LIN {X -82.2665,Y 110.2937,Z 192,A 113.0141,B 0.4199,C -0.1101,E1 0.3591,E2 342.9376} C_DIS
LIN {X -86.0435,Y 107.374,Z 192,A 114.6474,B 0.4204,C -0.1085,E1 0.3553,E2 341.3345} C_DIS
LIN {X -91.3683,Y 102.8804,Z 192,A 118.1809,B 0.4212,C -0.1052,E1 0.3472,E2 337.7503} C_DIS
LIN {X -95.472,Y 99.0842,Z 192,A 120.8102,B 0.4219,C -0.1023,E1 0.3415,E2 335.097} C_DIS
LIN {X -98.6871,Y 95.8821,Z 192,A 123.789,B 0.4227,C -0.0991,E1 0.3352,E2 332.0258} C_DIS
LIN {X -102.4573,Y 91.8421,Z 192,A 125.6577,B 0.4233,C -0.0962,E1 0.3315,E2 330.1958} C_DIS
LIN {X -105.4008,Y 88.4485,Z 192,A 128.4533,B 0.4241,C -0.0925,E1 0.3261,E2 327.3203} C_DIS
LIN {X -107.7268,Y 85.6004,Z 192,A 129.7733,B 0.4246,C -0.0904,E1 0.3237,E2 326.0198} C_DIS
LIN {X -110.5666,Y 81.9001,Z 192,A 132.1239,B 0.4254,C -0.0867,E1 0.3194,E2 323.6341} C_DIS
LIN {X -113.4298,Y 77.8855,Z 192,A 135.0925,B 0.4263,C -0.0819,E1 0.3143,E2 320.5837} C_DIS
LIN {X -115.9398,Y 74.0976,Z 192,A 137.5726,B 0.4271,C -0.0776,E1 0.3103,E2 318.0503} C_DIS
LIN {X -118.928,Y 69.2004,Z 192,A 140.7663,B 0.4281,C -0.0717,E1 0.3054,E2 314.7818} C_DIS
LIN {X -121.2848,Y 64.9809,Z 192,A 143.4167,B 0.429,C -0.0666,E1 0.3017,E2 312.071} C_DIS
LIN {X -123.0972,Y 61.4772,Z 192,A 145.4861,B 0.4296,C -0.0623,E1 0.2989,E2 309.9607} C_DIS
LIN {X -124.325,Y 58.9524,Z 192,A 147.1397,B 0.4301,C -0.0589,E1 0.2968,E2 308.2596} C_DIS
LIN {X -125.7064,Y 55.9456,Z 192,A 149.201,B 0.4307,C -0.0546,E1 0.2943,E2 306.1302} C_DIS
LIN {X -127.1851,Y 52.4996,Z 192,A 151.2785,B 0.4312,C -0.0501,E1 0.2919,E2 304.0008} C_DIS
LIN {X -128.3566,Y 49.5644,Z 192,A 153.2224,B 0.4317,C -0.0458,E1 0.2898,E2 301.9923} C_DIS
LIN {X -129.872,Y 45.4464,Z 192,A 155.8864,B 0.4323,C -0.0398,E1 0.2872,E2 299.2408} C_DIS
LIN {X -131.0593,Y 41.8977,Z 192,A 158.0817,B 0.4327,C -0.0346,E1 0.2852,E2 296.9778} C_DIS
LIN {X -132.1127,Y 38.448,Z 192,A 160.2392,B 0.4331,C -0.0295,E1 0.2834,E2 294.7494} C_DIS
LIN {X -133.0701,Y 34.9937,Z 192,A 162.521,B 0.4334,C -0.024,E1 0.2817,E2 292.3807} C_DIS
LIN {X -134.026,Y 31.1332,Z 192,A 165.1478,B 0.4338,C -0.0177,E1 0.2799,E2 289.6447} C_DIS
LIN {X -134.026,Y 31.1332,Z 192,A 165.1468,B 0.4338,C -0.0177,E1 0.2799,E2 289.6458} C_DIS
LIN {X -134.8958,Y 27.1154,Z 192,A 167.4299,B 0.434,C -0.0119,E1 0.2785,E2 287.2976} C_DIS
LIN {X -135.6359,Y 23.1335,Z 192,A 170.0281,B 0.434,C -0.0054,E1 0.2772,E2 284.5936} C_DIS
LIN {X -136.2319,Y 19.311,Z 192,A 172.3565,B 0.4341,C 0.0005,E1 0.2762,E2 282.1804} C_DIS
LIN {X -136.6496,Y 16.0924,Z 192,A 174.4138,B 0.4341,C 0.0058,E1 0.2755,E2 280.0384} C_DIS
LIN {X -137.0229,Y 12.5356,Z 192,A 176.8463,B 0.434,C 0.0119,E1 0.2748,E2 277.4908} C_DIS
LIN {X -137.0229,Y 12.5356,Z 192,A 176.8454,B 0.434,C 0.0119,E1 0.2748,E2 277.4919} C_DIS
LIN {X -137.3313,Y 8.4958,Z 192,A 179.2151,B 0.4337,C 0.0181,E1 0.2743,E2 275.0379} C_DIS
LIN {X -137.5082,Y 4.88,Z 192,A -178.5822,B 0.4335,C 0.0238,E1 0.274,E2 272.7481} C_DIS
LIN {X -137.5908,Y 1.0624,Z 192,A -176.18,B 0.4331,C 0.03,E1 0.274,E2 270.2427} C_DIS
LIN {X -137.5762,Y -2.2074,Z 192,A -173.9805,B 0.4327,C 0.0356,E1 0.274,E2 267.935} C_DIS
LIN {X -137.4523,Y -6.2721,Z 192,A -171.2346,B 0.432,C 0.0426,E1 0.2743,E2 265.051} C_DIS
LIN {X -137.4523,Y -6.2721,Z 192,A -171.2357,B 0.432,C 0.0426,E1 0.2743,E2 265.0522} C_DIS
LIN {X -137.1605,Y -10.9306,Z 192,A -168.4149,B 0.4312,C 0.0498,E1 0.2749,E2 262.1148} C_DIS
LIN {X -136.8034,Y -14.7268,Z 192,A -166.1744,B 0.4305,C 0.0555,E1 0.2756,E2 259.7865} C_DIS
LIN {X -136.3884,Y -18.1751,Z 192,A -163.8908,B 0.4298,C 0.0612,E1 0.2764,E2 257.3887} C_DIS
LIN {X -135.7544,Y -22.4235,Z 192,A -161.2462,B 0.4288,C 0.0678,E1 0.2776,E2 254.6261} C_DIS
LIN {X -135.1507,Y -25.8129,Z 192,A -159.1312,B 0.4279,C 0.0729,E1 0.2787,E2 252.416} C_DIS
LIN {X -134.4519,Y -29.2356,Z 192,A -157.0736,B 0.4271,C 0.0779,E1 0.28,E2 250.2736} C_DIS
LIN {X -133.7317,Y -32.3702,Z 192,A -155.0624,B 0.4262,C 0.0826,E1 0.2813,E2 248.167} C_DIS
LIN {X -132.8152,Y -35.9495,Z 192,A -152.8124,B 0.4251,C 0.0879,E1 0.283,E2 245.8152} C_DIS
LIN {X -131.7717,Y -39.6063,Z 192,A -150.3328,B 0.4239,C 0.0934,E1 0.2851,E2 243.2058} C_DIS
LIN {X -130.4308,Y -43.8167,Z 192,A -147.8826,B 0.4227,C 0.099,E1 0.2873,E2 240.6668} C_DIS
LIN {X -129.0421,Y -47.7534,Z 192,A -145.1723,B 0.4213,C 0.1047,E1 0.2901,E2 237.8131} C_DIS
LIN {X -127.4468,Y -51.8599,Z 192,A -142.8755,B 0.42,C 0.1096,E1 0.2926,E2 235.4479} C_DIS
LIN {X -125.9536,Y -55.3927,Z 192,A -140.6581,B 0.4188,C 0.1141,E1 0.2952,E2 233.1378} C_DIS
LIN {X -124.712,Y -58.1292,Z 192,A -138.9322,B 0.4179,C 0.1175,E1 0.2974,E2 231.3405} C_DIS
LIN {X -122.9457,Y -61.7801,Z 192,A -136.4951,B 0.4166,C 0.1221,E1 0.3006,E2 228.7902} C_DIS
LIN {X -118.9907,Y -69.0921,Z 192,A -132.2334,B 0.4142,C 0.13,E1 0.3067,E2 224.407} C_DIS
LIN {X -118.9907,Y -69.0921,Z 192,A -132.2343,B 0.4142,C 0.13,E1 0.3067,E2 224.4081} C_DIS
LIN {X -117.7679,Y -71.1561,Z 192,A -130.4987,B 0.4133,C 0.1327,E1 0.3095,E2 222.5591} C_DIS
LIN {X -115.1614,Y -75.3028,Z 192,A -127.9282,B 0.4119,C 0.137,E1 0.3136,E2 219.9066} C_DIS
LIN {X -112.6259,Y -79.0442,Z 192,A -125.5288,B 0.4107,C 0.1407,E1 0.3177,E2 217.4268} C_DIS
LIN {X -109.7298,Y -83.0172,Z 192,A -122.9996,B 0.4094,C 0.1444,E1 0.3223,E2 214.8225} C_DIS
LIN {X -107.0193,Y -86.4833,Z 192,A -120.7699,B 0.4083,C 0.1474,E1 0.3265,E2 212.5305} C_DIS
LIN {X -104.1301,Y -89.9412,Z 192,A -118.4564,B 0.4072,C 0.1504,E1 0.331,E2 210.1483} C_DIS
LIN {X -101.4439,Y -92.9605,Z 192,A -116.4182,B 0.4063,C 0.1528,E1 0.3351,E2 208.0539} C_DIS
LIN {X -98.3447,Y -96.2332,Z 192,A -114.1999,B 0.4054,C 0.1552,E1 0.3398,E2 205.7815} C_DIS
LIN {X -95.2449,Y -99.3023,Z 192,A -111.9693,B 0.4046,C 0.1574,E1 0.3447,E2 203.485} C_DIS
LIN {X -91.7358,Y -102.5525,Z 192,A -109.8256,B 0.4037,C 0.1595,E1 0.3494,E2 201.317} C_DIS
LIN {X -88.4041,Y -105.4381,Z 192,A -107.7408,B 0.403,C 0.1613,E1 0.3543,E2 199.1921} C_DIS
LIN {X -84.9501,Y -108.2402,Z 192,A -105.7485,B 0.4024,C 0.1629,E1 0.3589,E2 197.1773} C_DIS
LIN {X -81.8122,Y -110.6319,Z 192,A -103.772,B 0.4019,C 0.1641,E1 0.3638,E2 195.1471} C_DIS
LIN {X -77.3454,Y -113.7991,Z 192,A -101.3025,B 0.4013,C 0.1655,E1 0.3699,E2 192.6467} C_DIS
LIN {X -73.466,Y -116.341,Z 192,A -99.0682,B 0.401,C 0.1664,E1 0.3757,E2 190.3632} C_DIS
LIN {X -70.7312,Y -118.0241,Z 192,A -97.964,B 0.4006,C 0.1672,E1 0.3784,E2 189.2962} C_DIS
LIN {X -67.6259,Y -119.8302,Z 192,A -96.2319,B 0.4004,C 0.1676,E1 0.383,E2 187.5257} C_DIS
LIN {X -63.5638,Y -122.0318,Z 192,A -94.3513,B 0.4002,C 0.1683,E1 0.388,E2 185.6513} C_DIS
LIN {X -60.2882,Y -123.6838,Z 192,A -92.591,B 0.4002,C 0.1684,E1 0.3928,E2 183.8531} C_DIS
LIN {X -57.1515,Y -125.1641,Z 192,A -91.3146,B 0.4,C 0.1688,E1 0.3962,E2 182.6032} C_DIS
LIN {X -53.6848,Y -126.6901,Z 192,A -89.4231,B 0.4,C 0.1686,E1 0.4016,E2 180.6604} C_DIS
LIN {X -50.5881,Y -127.9586,Z 192,A -88.3401,B 0.3999,C 0.1689,E1 0.4045,E2 179.6268} C_DIS
LIN {X -47.9438,Y -128.9707,Z 192,A -87.1168,B 0.3999,C 0.1689,E1 0.4079,E2 178.3959} C_DIS
LIN {X -44.8741,Y -130.0704,Z 192,A -85.8215,B 0.3999,C 0.1688,E1 0.4116,E2 177.11} C_DIS
LIN {X -41.6562,Y -131.1364,Z 192,A -84.4103,B 0.4001,C 0.1685,E1 0.4156,E2 175.6981} C_DIS
LIN {X -38.5987,Y -132.0686,Z 192,A -83.1525,B 0.4001,C 0.1683,E1 0.4192,E2 174.4515} C_DIS
LIN {X -35.3952,Y -132.963,Z 192,A -81.8208,B 0.4003,C 0.1679,E1 0.423,E2 173.1276} C_DIS
LIN {X -32.2145,Y -133.7692,Z 192,A -80.468,B 0.4005,C 0.1675,E1 0.427,E2 171.7764} C_DIS
LIN {X -28.4913,Y -134.6126,Z 192,A -78.9786,B 0.4007,C 0.1669,E1 0.4313,E2 170.3021} C_DIS
LIN {X -22.8145,Y -135.6892,Z 192,A -76.9425,B 0.401,C 0.1663,E1 0.4371,E2 168.3242} C_DIS
LIN {X -16.8406,Y -136.5603,Z 192,A -74.2599,B 0.4018,C 0.1644,E1 0.4452,E2 165.6131} C_DIS
LIN {X -12.3791,Y -137.0377,Z 192,A -72.6307,B 0.4021,C 0.1635,E1 0.4499,E2 164.0211} C_DIS
LIN {X -8.5064,Y -137.3306,Z 192,A -71.1805,B 0.4025,C 0.1626,E1 0.4541,E2 162.5966} C_DIS
LIN {X -4.5589,Y -137.5199,Z 192,A -69.5432,B 0.4031,C 0.1612,E1 0.459,E2 160.9596} C_DIS
LIN {X -0.555,Y -137.593,Z 192,A -68.2325,B 0.4034,C 0.1604,E1 0.4627,E2 159.7049} C_DIS
Enddeposition()
END
